# B&R Automation Studio project ControlPLC_DataDistribution (part 5)

#### Main.st - Init, cyclic, exit code
```iecst
PROGRAM _INIT

	Name := 'Print Job Management';

	// Restore current print job management information from permanent memory.
	gPrintJobManagement.currentState := Nonvolatile;

	subscribePLCOpen( gPrintJobManagement.commands.updateLayerNumber, Name, task.command.updateCurrentLayer, task.internal.PLCOpen);

	subscribePLCOpen( gPrintJobManagement.commands.validatePrintFile, Name, task.command.validatePrintFile, task.internal.PLCOpen);

	subscribePLCOpen( gSystemRecipeApi.events.buildInfoLoaded, Name, task.command.validatePrintFile, task.internal.PLCOpen);
	subscribePLCOpen( gPrintJobManagement.commands.resetPrintInfo, Name, task.command.resetPrintInfo, task.internal.PLCOpen);

	registerStateBool( gPrintJobManagement.status.buildInfoValid, 'Build Info Loaded', task.status.buildInfoValid);

	//REASONS FOR INVALID BUILD FILE
	registerStateBool( gPrintJobManagement.status.buildInfoInvalid, 'Build Name Invalid', task.status.buildInfoInvalidReasons.invalidBuildName);
	registerStateBool( gPrintJobManagement.status.buildInfoInvalid, 'Num Layers Invalid', task.status.buildInfoInvalidReasons.invalidNumLayers);
	registerStateBool( gPrintJobManagement.status.buildInfoInvalid, 'Layer Height Invalid', task.status.buildInfoInvalidReasons.invalidLayerHeight);
	registerStateBool( gPrintJobManagement.status.buildInfoInvalid, 'Platform ID Invalid', task.status.buildInfoInvalidReasons.invalidPlatformID);
	registerStateBool( gPrintJobManagement.status.buildInfoInvalid, 'Machine Name Invalid', task.status.buildInfoInvalidReasons.invalidMachineName);
	registerStateBool( gPrintJobManagement.status.buildInfoInvalid, 'Pixel Map Ver. Invalid', task.status.buildInfoInvalidReasons.invalidPixelMapVersion);
	//registerStateBool( gPrintJobManagement.status.buildInfoInvalid, 'Pixel Usage Invalid', task.status.buildInfoInvalidReasons.invalidPixelUsage);

	//	registerStateBool( gPrintJobManagement.status.buildInfoInvalid, 'Workspace Boundaries Invalid', task.status.buildInfoInvalidReasons.invalidWorkspace);	 //TODO ADD BACK WHEN BUILD INFO FILE HAS THIS

	registerStateBool( gPrintJobManagement.status.buildInfoInvalid, 'PCI File Invalid', task.status.buildInfoInvalidReasons.invalidPrintConfigInstruction);

	gConfiguration.machineIdentity.machineName := 'DP12';
	gConfiguration.machineIdentity.machineNumber := 12;

	//SIM helper for bootup to set some non vol
	IF gSimulation THEN
		//gConfiguration.machineIdentity.factoryName := 'VulcanOne';
		//gConfiguration.machineIdentity.factoryNumber := FACTORY_VULCAN_ONE;
		//gConfiguration.machineIdentity.machineGeneration := MACHINE_GENERATION_GEN3;
			gConfiguration.machineIdentity.machineName := 'DP12';
		//gConfiguration.machineIdentity.machineType := MACHINE_TYPE_PRINTER;
		//	gConfiguration.machineIdentity.machineNumber := 13;

	END_IF

END_PROGRAM

PROGRAM _CYCLIC

	//Copy current state to non-volatile memory.
	Nonvolatile := gPrintJobManagement.currentState;
	dCurrentState ACCESS ADR(gPrintJobManagement.currentState);

	task.status.ready := TRUE;

	IF gSimulation THEN
		SimulateIO;
	END_IF
	/////////////////////////////////////////////////////////////////////////////////////////////////
	//COMMANDS
	//validate build info file
	//check if ready for printing
	//increment layer number

	//Cyclically this task also manages the part height and parameters related to the build info file
	/////////////////////////////////////////////////////////////////////////////////////////////////

	IF task.status.ready THEN

		IF task.internal.localLockout THEN

		ELSIF task.command.validatePrintFile THEN

			task.internal.newCommand := TRUE;
			task.status.statusMessage := 'Validating Build Info File';
			task.status.state := STATE_VALIDATING_BUILD_INFO;

		ELSIF task.command.updateCurrentLayer THEN

			task.internal.newCommand := TRUE;
			task.status.statusMessage := 'Updating Layer Number';
			task.status.state := STATE_UPDATE_LAYER_NUMBER;

		END_IF

	ELSE

		IF NOT allZero( ADR(task.command), SIZEOF(task.command)) THEN
			//vfAlarmEdgeSnippet(gPrintJobManagement.alarms.components, gPrintJobManagement.alarms.COMMAND_BEFORE_READY, 'Print Job Manager');
		END_IF

		task.internal.PLCOpen.status := PRINT_JOB_MANAGER_ERROR;
		task.status.state := STATE_NOT_READY;
		task.internal.localLockout := FALSE;

	END_IF

	///////////////////////////////////////////////////////////////
	// Handle any canceled commands that are required
	///////////////////////////////////////////////////////////////
	IF task.internal.newCommand THEN

		// TODO: Log state changes
		//		task.internal.abortedStep := task.status.sequence;
		//		task.internal.abortedState := task.internal.previousState;

		task.status.sequence := SEQUENCE_IDLE;

		// If a new command came into the system, abort any PLCOpen commands that were active.
		// If the command came from PLCOpen FirstPass will be true and it will not abort it
		atnPLCOpenAbort(task.internal.PLCOpen);

	END_IF

	CASE task.status.state OF

		STATE_NOT_READY:

			task.status.sequence := SEQUENCE_IDLE;

			task.status.statusMessage := 'Print job manager is not in ready state';

			IF task.status.ready THEN

				task.status.state := STATE_READY;

				task.status.statusMessage := 'Print job manager is in ready state';

			END_IF

		STATE_READY:

			task.status.sequence := SEQUENCE_IDLE;
			task.internal.localLockout := FALSE;

		STATE_RESETTING_PRINT_INFO:

			CASE task.status.sequence OF

				SEQUENCE_ERROR:
					task.status.statusMessage := 'Error resetting print data';

					//Handle Error
					task.internal.PLCOpen.status := PRINT_JOB_MANAGER_ERROR;
					task.status.state := STATE_READY;

				SEQUENCE_DONE:
					task.status.statusMessage := 'Print Data has been Reset';

					//Handle Done
					task.internal.PLCOpen.status := ERR_OK;
					task.status.state := STATE_READY;

				SEQUENCE_IDLE:

					task.status.statusMessage := 'Resetting Print Data';
					task.status.sequence := SEQUENCE_ABORT_DISTRIBUTION;

				ELSE

					ResetPrintInfoSubsequence;

			END_CASE

		STATE_UPDATE_LAYER_NUMBER:

			dCurrentState.currentLayerNumber := gPrintJobManagement.currentState.nextLayerNumber;

			Nonvolatile.currentLayerNumber := dCurrentState.currentLayerNumber;

			// Convert the current layer number to a string with the "nnnnn" format, adding required leading 0s.
			brsitoa(dCurrentState.currentLayerNumber, ADR(layerNumberValue_string));
			IF (dCurrentState.currentLayerNumber > 9999) THEN
				layerNumber_string := '';
			ELSIF (dCurrentState.currentLayerNumber > 999) THEN
				layerNumber_string := '0';
			ELSIF (dCurrentState.currentLayerNumber > 99) THEN
				layerNumber_string := '00';
			ELSIF (dCurrentState.currentLayerNumber > 9) THEN
				layerNumber_string := '000';
			ELSE
				layerNumber_string := '0000';
			END_IF
			brsstrcat(ADR(layerNumber_string), ADR(layerNumberValue_string));

			// Format the complete layer filename for the G-code (CNC) motion control file.
			layerFilename_GCode := Nonvolatile.baseFilename;
			brsstrcat(ADR(layerFilename_GCode), ADR('_L'));
			brsstrcat(ADR(layerFilename_GCode), ADR(layerNumber_string));
			brsstrcat(ADR(layerFilename_GCode), ADR('_GCode.cnc'));
			task.status.currentLayerGCodeFilename := layerFilename_GCode;

			task.internal.PLCOpen.status := ERR_OK;
			task.status.state := STATE_READY;

		STATE_VALIDATING_BUILD_INFO:

			CASE task.status.sequence OF

				SEQUENCE_ERROR:
					task.status.statusMessage := 'Error Validating Print Files';

					//Handle Error
					task.internal.PLCOpen.status := PRINT_JOB_MANAGER_ERROR;
					task.status.state := STATE_READY;

				SEQUENCE_DONE:
					task.status.statusMessage := 'Validating Print files finished';
					gPrintJobManagement.status.buildInfoValidCheck := TRUE;
					//Handle Done
					task.internal.PLCOpen.status := ERR_OK;
					task.status.state := STATE_READY;

				SEQUENCE_IDLE:

					task.status.statusMessage := 'Print File validation started';
					task.status.sequence := SEQUENCE_READ_BUILD_INFO;

				ELSE

					ValidateBuildFileSubsequence;
			END_CASE

	END_CASE

	//get reason that might occur outside of the sequence
	task.status.buildInfoError := stateTrueStatus( gPrintJobManagement.status.buildInfoInvalid, ADR( task.status.buildInfoErrorStatus ), SIZEOF(task.status.buildInfoErrorStatus));

	//---------------------------------------------------------------------------
	// Repopulate layer gcode file name if PLC restarted.
	//---------------------------------------------------------------------------

	IF (task.status.currentLayerGCodeFilename = '')  THEN

		// Convert the current layer number to a string with the "nnnnn" format, adding required leading 0s.
		brsitoa(dCurrentState.currentLayerNumber, ADR(layerNumberValue_string));
		IF (dCurrentState.currentLayerNumber > 9999) THEN
			layerNumber_string := '';
		ELSIF (dCurrentState.currentLayerNumber > 999) THEN
			layerNumber_string := '0';
		ELSIF (dCurrentState.currentLayerNumber > 99) THEN
			layerNumber_string := '00';
		ELSIF (dCurrentState.currentLayerNumber > 9) THEN
			layerNumber_string := '000';
		ELSE
			layerNumber_string := '0000';
		END_IF
		brsstrcat(ADR(layerNumber_string), ADR(layerNumberValue_string));

		// Format the complete layer filename for the G-code (CNC) motion control file.
		layerFilename_GCode := Nonvolatile.baseFilename;
		brsstrcat(ADR(layerFilename_GCode), ADR('_L'));
		brsstrcat(ADR(layerFilename_GCode), ADR(layerNumber_string));
		brsstrcat(ADR(layerFilename_GCode), ADR('_GCode.cnc'));
		task.status.currentLayerGCodeFilename := layerFilename_GCode;

	END_IF

	//RESET COMMANDS
	brsmemset(ADR(task.command), 0, SIZEOF(task.command));
	task.internal.newCommand := FALSE;

	task.internal.newCommand := 0;

	command();
	IF command.Done OR command.Error OR command.Aborted THEN
		command.Execute := FALSE;
	END_IF

	logStateChange_0.LoggerName := 'App';
	logStateChange_0.ModuleName := Name;
	logStateChange_0.State 		:= task.status.state;
	logStateChange_0.StateName 	:= task.status.statusMessage;
	logStateChange_0();

	logSeqChange_0.LoggerName 	:= 'App';
	logSeqChange_0.ModuleName 	:= Name;
	//	logSeqChange_0.State		:= task.status.sequence;
	//	logSeqChange_0.StateName	:= task.status.statusMessage;
	//	logSeqChange_0();

	// ---------------------------------------------------------------------------
	// Call ATN FUB
	// ---------------------------------------------------------------------------

	//task.status.buildInfoValid := stateAllFalse( gPrintJobManagement.status.buildInfoInvalid, TRUE);

	gPrintJobManagement.status.currentLayerGCodeFilename := task.status.currentLayerGCodeFilename;

END_PROGRAM

PROGRAM _EXIT

END_PROGRAM
```

#### Types.typ - Local data types
```iecst
TYPE
	test_typ : 	STRUCT
		command : testCommand_typ;
	END_STRUCT;
	testCommand_typ : 	STRUCT
		induceCurrentLayerToEleven : BOOL;
		assertDOMS : BOOL;
		assertRegularPlate : BOOL;
	END_STRUCT;
	Configuration_typ : 	STRUCT
		BUILD_PLATE_THICKNESS_MAX_MM : REAL;
		BLADE_OFFSET_MAX_MM : REAL;
		FOCAL_OFFSET_MAX_MM : REAL;
		FOCAL_OFFSET_MIN_MM : REAL;
		FOCAL_OFFSET_MM : REAL;
		OPTICS_BOX_REVISION : USINT;
		BLADE_OFFSET_MM : REAL;
		ENCODER_TICK_WIDTH : REAL;
		MAX_LASER_COUNT : UINT;
		LASER_LINE_ANGLE : REAL;
		HEAD_CENTER_OFFSET : REAL;
		LASER_SPACING : REAL;
		MIN_LASER_WATTS : REAL;
		MAX_LASER_WATTS : REAL;
	END_STRUCT;
	IO_typ : 	STRUCT
		_ : USINT;
	END_STRUCT;
	localInterface_typ : 	STRUCT
		command : localInterfaceCommand_typ;
		parameters : localInterfaceParameter_typ;
		status : localInterfaceStatus_typ;
		internal : localInterfaceInternal_typ;
	END_STRUCT;
	localInterfaceCommand_typ : 	STRUCT
		updateCurrentLayer : BOOL;
		validatePrintFile : BOOL;
		checkReadyForPrinting : BOOL;
		resetLayerNumberToZero : BOOL;
		restartAtSpecifiedLayer : BOOL;
		setBuildPlateThickness : BOOL;
		setFocalOffset : BOOL;
		publishConfigurationData : BOOL;
		setRecoaterOffset : BOOL;
		resetPrintInfo : BOOL;
		bladeOffsetClr : BOOL;
		bladeOffsetPlusTen : BOOL;
		bladeOffsetMinusTen : BOOL;
		setThicknessDOMS : BOOL;
		clearThicknessDOMS : BOOL;
		resetPlateType : BOOL;
		enableLOP : BOOL;
		disableLOP : BOOL;
		calculateRemainingPrintTime : BOOL;
		coolingDelay : BOOL;
	END_STRUCT;
	localInterfaceParameter_typ : 	STRUCT
		layerToDistribute : UINT;
		printJobLayer : UINT;
		startingLayerNumber : UDINT;
	END_STRUCT;
	localInterfaceInternal_typ : 	STRUCT
		PLCOpenConfigData : AtnPlcOpenStatus;
		PLCOpen : AtnPlcOpenStatus;
		checkPixelUsage : AtnPLCOpen;
		previousState : STATE;
		newCommand : BOOL;
		localLockout : BOOL;
		subSystemStatus : ARRAY[0..10]OF STRING[80];
		remapPixels : AtnPLCOpen;
	END_STRUCT;
	localInterfaceStatus_typ : 	STRUCT
		currentLayerGCodeFilename : STRING[255];
		recoaterOffsetInvalid : BOOL;
		focalOffset : REAL;
		recoaterOffset : REAL;
		buildPlateThicknessInvalid : BOOL;
		buildPlateThickness : REAL;
		buildInfoValid : BOOL;
		buildInfoNotInvalid : BOOL;
		buildInfoError : BOOL;
		distributionTimeout : BOOL;
		buildInfoErrorStatus : ARRAY[0..19]OF STRING[80];
		ready : BOOL;
		sequence : SEQUENCE;
		statusMessage : STRING[vfALARMS_MAX_SNIPPET_STR_LENGTH];
		state : STATE;
		buildInfoInvalidReasons : buildInfoInvalidReasons_typ;
	END_STRUCT;
	SEQUENCE :
		(
		SEQUENCE_IDLE,
		SEQUENCE_DONE,
		SEQUENCE_ERROR,
		SEQUENCE_READ_BUILD_INFO,
		SEQUENCE_CHECK_PIXEL_USAGE,
		SEQUENCE_DO_PIXEL_MAP,
		SEQUENCE_CHECK_LASERS,
		SEQUENCE_CHECK_PUMPS,
		SEQUENCE_CHECK_O2_LEVELS,
		SEQUENCE_CHECK_PNEUMATIC_SUPPLY,
		SEQUENCE_CHECK_AXES_STATE,
		SEQUENCE_CHECK_RECOATER_POS,
		SEQUENCE_CHECK_LIFT_POS,
		SEQUENCE_CHECK_LAYER_NUMBER,
		SEQUENCE_CHECK_CAMERA,
		SEQUENCE_ASK_IF_OK_TO_RESET,
		SEQUENCE_CLEAR_DATA,
		SEQUENCE_ABORT_DISTRIBUTION
		);
	STATE :
		(
		STATE_READY,
		STATE_NOT_READY,
		STATE_CHECKING_PRINT_READY,
		STATE_UPDATE_LAYER_NUMBER,
		STATE_VALIDATING_BUILD_INFO,
		STATE_SET_BUILD_PLATE_THICKNESS,
		STATE_COOLING_DELAY,
		STATE_SET_FOCAL_OFFSET,
		STATE_SET_DOMS_THICKNESS,
		STATE_SET_RECOATER_OFFSET,
		STATE_RESETTING_PRINT_INFO,
		STATE_ERROR
		);
	buildInfoInvalidReasons_typ : 	STRUCT
		invalidPixelUsage : BOOL;
		invalidPixelMapVersion : BOOL;
		invalidMachineName : BOOL;
		invalidPlatformID : BOOL;
		invalidLayerHeight : BOOL;
		invalidNumLayers : BOOL;
		invalidBuildName : BOOL;
		invalidToolpath : BOOL;
		invalidWorkspace : BOOL;
		invalidPlateOrigin : BOOL;
		invalidPrintConfigInstruction : BOOL;
	END_STRUCT;
END_TYPE
```

#### SubSequence.st
```iecst
ACTION ValidateBuildFileSubsequence:

	CASE task.status.sequence OF

		SEQUENCE_READ_BUILD_INFO:

			task.status.statusMessage := 'Checking build info contents';

			// NOTES:====================================================
			// base_filename must be 13 charaters long (e.g. VF-00001-0001)
			// build_layout and print_number must be > 0
			// num_layers must be > 0
			// layer_height must be within established range
			// PLATFORM_MEDIUM_400x600 is not currently supported
			// PrinterInfo.name must match the machineIdentity.machineName setting

			task.status.buildInfoInvalidReasons.invalidBuildName := (gBuildInformation.build_layout = 0) OR (gBuildInformation.print_number = 0) OR (brsstrlen(ADR(gBuildInformation.base_filename)) <> 13);
			task.status.buildInfoInvalidReasons.invalidNumLayers := (gBuildInformation.num_layers = 0);
			task.status.buildInfoInvalidReasons.invalidLayerHeight := (gBuildInformation.layer_height < MIN_LAYER_HEIGHT) OR (gBuildInformation.layer_height > MAX_LAYER_HEIGHT);
			task.status.buildInfoInvalidReasons.invalidPlatformID := (gBuildInformation.platform_id <> PLATFORM_SMALL_200x600) AND (gBuildInformation.platform_id <> PLATFORM_LARGE_600x600);
			task.status.buildInfoInvalidReasons.invalidMachineName := (brsstrcmp(ADR(gBuildInformation.BuildInstanceInfo.PrinterInfo.name), ADR(gConfiguration.machineIdentity.machineName)) <> 0);

			//task.status.buildInfoInvalidReasons.invalidPrintConfigInstruction := NOT(gPrintProcessConfig.MachineName = gConfiguration.machineIdentity.machineName) OR NOT(gPrintProcessConfig.FileFormatVersion = gPrintJobManagement.currentState.PCIFileFormatVersion);

			//because if nothing exists in nonvolatile then this will never work
			IF Nonvolatile.pixelMapFileVersion = 0 THEN
				Nonvolatile.pixelMapFileVersion := 1;
			END_IF

				task.status.buildInfoValid := TRUE;
				gPrintJobManagement.currentState.buildInfoCheckValid := task.status.buildInfoValid;
				// If the BuildInfo file is different from the one that was previously running, reset to layer zero to start a new print.
				(*	IF (gBuildInformation.build_layout <> dCurrentState.buildLayout)
				OR (gBuildInformation.print_number <> dCurrentState.printNumber)
				OR (gBuildInformation.layer_height <> dCurrentState.layerHeight) THEN

				task.command.resetLayerNumberToZero := TRUE;//todo
				ELSE *)

				//populate print info
				dCurrentState.baseFilename := gBuildInformation.base_filename;
				dCurrentState.buildIteration := gBuildInformation.build_iter;
				dCurrentState.buildLayout := gBuildInformation.build_layout;
				dCurrentState.printNumber := gBuildInformation.print_number;
				dCurrentState.numberOfLayers := gBuildInformation.num_layers;
				dCurrentState.layerHeight := gBuildInformation.layer_height;
				//dCurrentState.buildPlatform := PLATFORM_LARGE_600x600;//fixed value ignore BD
				dCurrentState.description := gBuildInformation.description;
				dCurrentState.author := gBuildInformation.author;
				dCurrentState.printOwner := gBuildInformation.print_owner;

				task.status.sequence := SEQUENCE_DONE;

	END_CASE

END_ACTION

ACTION ResetPrintInfoSubsequence:

	CASE task.status.sequence OF

		SEQUENCE_ABORT_DISTRIBUTION:

			executeCommand(gBuildDistributorApi.commands.abortDistribution);
			task.status.sequence := SEQUENCE_CLEAR_DATA;

		SEQUENCE_CLEAR_DATA:

			task.status.sequence := SEQUENCE_DONE;
	END_CASE

	END_ACTION
```

#### Simulation.st
```iecst
ACTION SimulateIO:

	//used in the electrode test case -> electrode only enable if layer 10 or more
	IF test.command.induceCurrentLayerToEleven THEN
		test.command.induceCurrentLayerToEleven := FALSE;
		gPrintJobManagement.currentState.currentLayerNumber := 11;
		gPrintJobManagement.currentState.lastPrintedLayerNumber := 10;
		gPrintJobManagement.currentState.lastRecoatedLayerNumber := 10;
	END_IF

END_ACTION
```

### Program Logical/DataManagement/PrintJobManagement/BuildDistributor (IEC)

#### Main.st - Init, cyclic, exit code
```iecst
PROGRAM _INIT

	Name := 'Build Distributor';

	//direct commands to operate the chiller
	subscribePLCOpenWithParameters ( gBuildDistributorApi.commands.startDistribution, Name, ADR(task.parameters.layerNumberToDistribute), SIZEOF(task.parameters.layerNumberToDistribute), task.command.startDistribution, task.internal.PLCOpen);
	subscribePLCOpen( gBuildDistributorApi.commands.distributeLayerFile, Name, task.command.distributeLayerFile, task.internal.PLCOpen );
	subscribePLCOpenWithParameters ( gBuildDistributorApi.commands.abortDistribution, Name, 0, 0, task.command.abortDistribution, task.internal.PLCOpen);

	//other systems can monitor this state
	registerStateBool( gBuildDistributorApi.status.subsystemsReady, Name, task.status.buildDistributorConnected);

END_PROGRAM

PROGRAM _CYCLIC

	//Call piper interface
	PiperModuleInterface;

	///////////////////////////////////////////////////////////////
	//API:
	//	Requires:
	//	-
	//	Commands:
	//	-takePrescan
	//	-takePostscan
	//  -takeManual
	//	Inhbits:
	//	-

	//  State Monitoring
	//  -
	///////////////////////////////////////////////////////////////

	//Heartbeat set and monitor
	task.internal.heartbeatTimer.PT := T#1s;
	task.internal.heartbeatTimer.IN := NOT(task.internal.heartbeatTimer.Q);
	IF (task.internal.heartbeatTimer.Q) THEN
		gOpcData_ToBuildPC.Heartbeat := gOpcData_ToBuildPC.Heartbeat + 1;
		IF (gOpcData_FromBuildPC.Heartbeat <> task.internal.lastHeartbeatReceived) THEN
			task.internal.lastHeartbeatReceived := gOpcData_FromBuildPC.Heartbeat;
			task.status.buildDistributorConnected := TRUE;
			task.status.missedHeartbeats := 0;
		ELSE
			task.status.missedHeartbeats := task.status.missedHeartbeats + 1;
		END_IF
	END_IF
	task.internal.heartbeatTimer();

	//timeout after 3 missed heartbeats
	IF task.status.missedHeartbeats > 10 THEN
		task.status.buildDistributorConnected := FALSE;
	END_IF

	//Reset signals if data distributor disconnects
	IF NOT(task.status.buildDistributorConnected) THEN
		gOpcData_ToBuildPC.RequestAbortDistribution := FALSE;
		gOpcData_ToBuildPC.RequestPauseDistribution := FALSE;
		gOpcData_ToBuildPC.RequestStartDistribution := FALSE;
		gOpcData_ToBuildPC.PrintingActive := FALSE;
		gOpcData_ToBuildPC.RequestBuildInfo := FALSE;
	END_IF

	//ADD LATER TODO
	//	vfAlarmPersistent(gVisionApi.alarms.components, gVisionApi.alarms.VISION_HEARTBEAT_LOST_AL1200, NOT(task.status.visionAppConnected));

	//ready to handle commands
	task.status.ready := stateTrueStatus( gBuildDistributorApi.status.subsystemsReady, ADR(task.internal.subSystemStatus), SIZEOF(task.internal.subSystemStatus) );

	IF NOT task.status.ready THEN
		stateStatus( gBuildDistributorApi.status.subsystemsReady, ADR(task.internal.subSystemStatus), SIZEOF(task.internal.subSystemStatus) );
	ELSE
		task.internal.subSystemStatus[0] := 'Ready';
	END_IF

	///////////////////////////////////////////////////////////////
	//Handle interpreting commands that do not require STATE_READY
	///////////////////////////////////////////////////////////////
	IF task.status.ready THEN

		//NOTE: Commands that just turn ON/OFF IO CAN happen in the command translation
		IF task.command.startDistribution THEN
			task.internal.newCommand := 1;

			task.status.sequence := SEQUENCE_IDLE;
			task.status.state := STATE_START_DISTRIBUTION;
			task.status.statusMessage := 'Starting Distribution';

		ELSIF task.command.distributeLayerFile THEN
			task.internal.newCommand := 1;
			task.status.sequence := SEQUENCE_IDLE;
			task.status.state := STATE_DISTRIBUTE_LAYER_FILE;
			task.status.statusMessage := 'Distributing Layer File';

		ELSIF task.command.abortDistribution THEN
			task.internal.newCommand := 1;
			task.status.sequence := SEQUENCE_IDLE;
			task.status.state := STATE_ABORT_DISTRIBUTION;
			task.status.statusMessage := 'Aborting Distribution';

		END_IF

	ELSE
		task.internal.PLCOpen.status := BUILD_DISTRIBUTOR_ERROR;
		task.status.state := STATE_NOT_READY;
		task.internal.localLockout := FALSE;
	END_IF

	///////////////////////////////////////////////////////////////
	//Handle any canceled commands that are required
	///////////////////////////////////////////////////////////////
	IF task.internal.newCommand THEN

		//TODO: Log state changes
		//		task.internal.abortedStep := task.status.sequence;
		//		task.internal.abortedState := task.internal.previousState;

		//If a new command came into the system, abort any PLCOpen commands that were active.
		// If the command came from PLCOpen FirstPass will be true and it will not abort it
		atnPLCOpenAbort(task.internal.PLCOpen);

	END_IF

	///////////////////////////////////////////////////////////////
	//Handle any Commands that do not require state.
	///////////////////////////////////////////////////////////////

	///////////////////////////////////////////////////////////////
	//Handle the current state
	///////////////////////////////////////////////////////////////
	CASE task.status.state OF

		STATE_NOT_READY:

			task.status.sequence := SEQUENCE_IDLE;
			task.status.statusMessage := 'Build Distributor is NOT ready';
			gOpcData_ToBuildPC.RequestBuildInfo := FALSE;

			IF task.status.ready THEN
				task.status.state := STATE_READY;
				task.status.statusMessage := 'Build Distributor is ready';
			END_IF

		STATE_READY:

			task.status.sequence := SEQUENCE_IDLE;
			task.internal.localLockout := FALSE;
			gOpcData_ToBuildPC.RequestBuildInfo := FALSE;

		STATE_START_DISTRIBUTION:

			CASE task.status.sequence OF

				SEQUENCE_ERROR:
					task.status.statusMessage := 'Start Distribution ERROR';
					task.internal.PLCOpen.status := BUILD_DISTRIBUTOR_ERROR;
					task.status.state := STATE_READY;

				SEQUENCE_DONE:
					task.status.statusMessage := 'Start Distribution COMPLETE';
					task.internal.PLCOpen.status := ERR_OK;
					task.status.state := STATE_READY;

				SEQUENCE_IDLE:
					task.status.statusMessage := 'Start Distribution busy...';
					task.status.sequence := SEQUENCE_EXECUTE_START_DIST;

				ELSE

					StartDistributionSubSequence;

			END_CASE

		STATE_DISTRIBUTE_LAYER_FILE:

			CASE task.status.sequence OF

				SEQUENCE_ERROR:
					task.status.statusMessage := 'Distribute Layer ERROR';
					task.internal.PLCOpen.status := BUILD_DISTRIBUTOR_ERROR;
					task.status.state := STATE_READY;

				SEQUENCE_DONE:
					task.status.statusMessage := 'Distribute Layer COMPLETE';
					task.internal.PLCOpen.status := ERR_OK;
					task.status.state := STATE_READY;

				SEQUENCE_IDLE:
					task.status.statusMessage := 'Distribute Layer busy...';
					task.status.sequence := SEQUENCE_EXECUTE_GET_LAYER_FILES;

				ELSE

					DistributeLayerFileSubSequence;

			END_CASE

		STATE_ABORT_DISTRIBUTION:

			task.status.statusMessage := 'aborting distribution';

			IF task.status.buildDistributorConnected THEN
				//gPrint Job management files
				gOpcData_ToBuildPC.RequestAbortDistribution := TRUE;
				gOpcData_ToBuildPC.RequestPauseDistribution := FALSE;
				gOpcData_ToBuildPC.RequestStartDistribution := FALSE;
				gOpcData_ToBuildPC.PrintingActive := FALSE;
				gOpcData_ToBuildPC.RequestBuildInfo := FALSE;

				IF (gOpcData_FromBuildPC.DistributionAborted) THEN
					gOpcData_ToBuildPC.RequestAbortDistribution := FALSE;

					//brsmemset( ADR(gPrintProcessConfig), 0, SIZEOF(gPrintProcessConfig) ); Not deleting. Keep last know value on Abort
					gPrintProcessConfigLoaded := FALSE;

					task.status.statusMessage := 'aborting complete';
					task.internal.PLCOpen.status := ERR_OK;
					task.status.state := STATE_READY;

				END_IF

			ELSE
				task.status.statusMessage := 'BD not connected';
				gOpcData_ToBuildPC.RequestAbortDistribution := FALSE;
				task.status.state := STATE_READY;
				task.internal.PLCOpen.status := ERR_OK;

			END_IF

	END_CASE

	///////////////////////////////////////////////////////////////
	//Update Statuses
	///////////////////////////////////////////////////////////////

	///////////////////////////////////////////////////////////////
	//Call all PLCOpen function blocks
	///////////////////////////////////////////////////////////////
	task.internal.fbTON_DistributionDelay();
	task.internal.fbTON_DistributionDelay.IN := FALSE;

	task.internal.atnPLCOpenCommand();
	task.internal.atnPLCOpenCommand.Execute := FALSE;

	task.internal.atnPLCOpenCommandParameters();
	task.internal.atnPLCOpenCommandParameters.Execute := FALSE;

	task.internal.distributorTimeout();
	task.internal.distributorTimeout.IN := FALSE;

	task.internal.distributionRecoveryTimer();
	task.internal.distributionRecoveryTimer.IN := FALSE;

	///////////////////////////////////////////////////////////////
	//Reset all commands to ensure they don't get buffered
	///////////////////////////////////////////////////////////////
	task.command.distributeLayerFile := 0;
	task.command.startDistribution := 0;
	task.command.abortDistribution := 0;
	task.internal.newCommand := 0;

	task.internal.waitToRetry();
	task.internal.waitToRetry.IN := FALSE;

	logStateChange_0.LoggerName := 'App';
	logStateChange_0.ModuleName := Name;
	logStateChange_0.State 		:= task.status.state;
	logStateChange_0.StateName 	:= task.status.statusMessage;
	logStateChange_0();

	logSeqChange_0.LoggerName 	:= 'App';
	logSeqChange_0.ModuleName 	:= Name;
	logSeqChange_0.State		:= task.status.sequence;
	logSeqChange_0.StateName	:= task.status.statusMessage;
	logSeqChange_0();

	//Keep track of the previous state
	task.internal.previousState := task.status.state;

	///////////////////////////////////////////////////////////////
	//Simulation
	///////////////////////////////////////////////////////////////
	IF gSimulation THEN
		SimulateIO;
	END_IF

END_PROGRAM

PROGRAM _EXIT
		(* Insert code here *)

END_PROGRAM
```

#### PiperInterface.st
```iecst
ACTION PiperModuleInterface:

	//Give this module a name so it is easier to debug
	ModuleInterface.ModuleName:=	Name;

	//Add a module to the Piper
	Module.ModuleInterface:=	ADR(ModuleInterface);
	Module.Piper:= 	ADR(gMachine);
	Module();

	// Handle any machine states that this module needs to respond to
	CASE ModuleInterface.PiperState OF
//		MACH_ST_BOOTING:
//		MACH_ST_CLEARING:
//		MACH_ST_STOPPED:
		MACH_ST_STARTING:

			ModuleInterface.ModuleResponse:=	ModuleInterface.PiperState;

			(*//sample piper integration

			//for when sequence is required for substate transition
			CASE ModuleInterface.PiperSubState OF

				0:

					//only need the chiller for printing but not other operations
					CASE gMachineState.operation OF

						MACHINE_OPERATIONS_PRINT_LAYER:
							ModuleInterface.ModuleSubStateRequest := SUB_STATE_CHECK_CHILLER;

						ELSE
							ModuleInterface.ModuleResponse:=	ModuleInterface.PiperState;

					END_CASE

				SUB_STATE_CHECK_CHILLER:

					//should be an edge command
					task.command.startChiller := TRUE;

					ModuleInterface.ModuleStatus := 'waiting chiller';

					IF task.status.chillerIsRunning THEN
						ModuleInterface.ModuleResponse:=	ModuleInterface.PiperState;
					END_IF

			END_CASE

			*)

//		MACH_ST_IDLE:
//		MACH_ST_SUSPENDED:
//		MACH_ST_EXECUTE:
//		MACH_ST_STOPPING:
//		MACH_ST_ABORTING:
//		MACH_ST_ABORTED:
//		MACH_ST_HOLDING:
//		MACH_ST_HELD:
//		MACH_ST_UNHOLDING:
//		MACH_ST_SUSPENDING:
//		MACH_ST_UNSUSPENDING:
//		MACH_ST_RESETTING:
//		MACH_ST_COMPLETING:
//		MACH_ST_COMPLETE:

		MACH_ST_BYPASSED:

		ELSE
			ModuleInterface.ModuleResponse:=	ModuleInterface.PiperState;

	END_CASE

	//for turning commands to edges to work with piper
	(*
	//Turn level commands to edges
	EdgePosArray( ADR(piperCommands), ADR(_piperCommands), ADR(task.command), SIZEOF(task.command) );
	brsmemset( ADR(piperCommands), 0, SIZEOF(piperCommands) );
	*)

END_ACTION
```

#### SubSequence.st
```iecst
// Start connection to build distributor and distribute the starting files
ACTION StartDistributionSubSequence:

	CASE task.status.sequence OF

		SEQUENCE_EXECUTE_START_DIST:

			task.status.sequence := SEQUENCE_REQUEST_BUILD_INFO;

		SEQUENCE_REQUEST_BUILD_INFO:

			task.status.statusMessage := 'ask for build info file';

			//gPrint Job management files
			gOpcData_ToBuildPC.RequestAbortDistribution := FALSE;
			gOpcData_ToBuildPC.RequestPauseDistribution := FALSE;
			gOpcData_ToBuildPC.RequestStartDistribution := FALSE;
			gOpcData_ToBuildPC.PrintingActive := FALSE;
			gOpcData_ToBuildPC.RequestBuildInfo := TRUE;

			//load the last file you had saved, if its 0 get layer 1
			gOpcData_ToBuildPC.CurrentPrintLayer := gPrintJobManagement.currentState.currentLayerNumber;
			IF (gOpcData_ToBuildPC.CurrentPrintLayer = 0) THEN
				gOpcData_ToBuildPC.CurrentPrintLayer := 1;
			END_IF

			task.status.sequence := SEQUENCE_BUILD_INFO_READY;

		SEQUENCE_BUILD_INFO_READY:

			IF (gOpcData_FromBuildPC.BuildInfoReady) THEN
				gOpcData_ToBuildPC.RequestBuildInfo := FALSE;
				task.status.sequence := SEQUENCE_LOAD_PCI_FILE;
			END_IF

		SEQUENCE_LOAD_PCI_FILE:

			task.status.statusMessage := 'Loading PCI File and Verifying';

			task.internal.atnPLCOpenCommand.Command := gSystemRecipeApi.commands.loadPrintProcessConfigFile;
			task.internal.atnPLCOpenCommand.Execute := TRUE;

			IF task.internal.atnPLCOpenCommand.Done OR gPrintJobManagement.status.loadPCIFileComplete THEN
				task.status.sequence := SEQUENCE_LOAD_BUILD_FILE;
				task.internal.atnPLCOpenCommand.Execute := FALSE;
				gPrintJobManagement.status.loadPCIFileComplete := FALSE;

			ELSIF task.internal.atnPLCOpenCommand.Error THEN
				task.status.sequence := SEQUENCE_ERROR;
			END_IF

		SEQUENCE_LOAD_BUILD_FILE:
			task.status.statusMessage := 'load build info file';
			task.internal.atnPLCOpenCommand.Command := gSystemRecipeApi.commands.loadBuildInfo;
			task.internal.atnPLCOpenCommand.Execute := TRUE;

			IF task.internal.atnPLCOpenCommand.Done OR gSystemRecipeApi.status.buildInfoLoaded THEN
				task.status.sequence := SEQUENCE_CHK_BUILD_INFO_VALID;
				gSystemRecipeApi.status.buildInfoLoaded := FALSE;
				task.internal.atnPLCOpenCommand.Execute := FALSE;

			ELSIF task.internal.atnPLCOpenCommand.Error THEN
				task.status.sequence := SEQUENCE_ERROR;
			END_IF

		SEQUENCE_CHK_BUILD_INFO_VALID:
			task.status.statusMessage := 'validating build info contents';
			task.internal.atnPLCOpenCommand.Command := gPrintJobManagement.commands.validatePrintFile;
			task.internal.atnPLCOpenCommand.Execute := TRUE;

			IF task.internal.atnPLCOpenCommand.Done OR gPrintJobManagement.status.buildInfoValidCheck THEN
				task.status.sequence := SEQUENCE_DELETE_LASER_FILES;
				gPrintJobManagement.status.buildInfoValidCheck:= FALSE;
				task.internal.atnPLCOpenCommand.Execute := FALSE;
				gPrintProcessConfigLoaded := TRUE; // Set flag after validating PCI with BuildInfo File
			ELSIF task.internal.atnPLCOpenCommand.Error THEN
				task.status.sequence := SEQUENCE_ERROR;
			END_IF

		SEQUENCE_DELETE_LASER_FILES:
			task.status.statusMessage := 'delete laser files';
			task.internal.atnPLCOpenCommand.Command := gVFLCR.command.deleteLaserControlFiles;
			task.internal.atnPLCOpenCommand.Execute := TRUE;

			IF task.internal.atnPLCOpenCommand.Done THEN
				task.status.sequence := SEQUENCE_START_DISTRIBUTION;
				task.internal.atnPLCOpenCommand.Execute := FALSE;
			ELSIF task.internal.atnPLCOpenCommand.Error THEN
				task.status.sequence := SEQUENCE_ERROR;
			END_IF

		SEQUENCE_START_DISTRIBUTION:
			task.status.statusMessage := 'distribute laser files';

			gOpcData_ToBuildPC.RequestStartDistribution := TRUE;
			task.status.sequence := SEQUENCE_VERIFY_DISTRIBUTION;

		SEQUENCE_VERIFY_DISTRIBUTION:

			task.status.statusMessage := 'verifying distribution';

			IF (gOpcData_FromBuildPC.CurrentDistributionLayer = gOpcData_ToBuildPC.CurrentPrintLayer) THEN

				task.internal.lastDistributedLayerNumber := UDINT_TO_UINT(gOpcData_ToBuildPC.CurrentPrintLayer);
				gPrintJobManagement.currentState.lastDistributedLayer := task.internal.lastDistributedLayerNumber;

				task.status.sequence := SEQUENCE_SET_CURRENT_LAYER;

			END_IF

			task.internal.distributorTimeout.PT := T#30s;
			task.internal.distributorTimeout.IN := TRUE;

			IF task.internal.distributorTimeout.Q THEN
				task.status.sequence := SEQUENCE_ERROR;
			END_IF

		SEQUENCE_SET_CURRENT_LAYER:

			//this is redundant, but that command also will re-set the CNC file name
			task.status.statusMessage := 'update current layer';

			//NOT NEEDED!
			Nonvolatile.currentLayerNumber := gPrintJobManagement.currentState.currentLayerNumber;

			task.status.sequence := SEQUENCE_DISTRIBUTION_STARTED;

		SEQUENCE_DISTRIBUTION_STARTED:
			gPrintJobManagement.currentState.newBuildInfoFileLoaded := TRUE;//TODO this should be set outside?
			task.status.sequence := SEQUENCE_DONE;
	END_CASE

END_ACTION

// Distribute Layer Files to VFLCR and adjust number
ACTION DistributeLayerFileSubSequence:

	CASE task.status.sequence OF

		SEQUENCE_EXECUTE_GET_LAYER_FILES:
			task.status.sequence := SEQUENCE_SET_DESIRED_LAYER;

		SEQUENCE_CHK_BUILD_INFO:
			task.status.statusMessage := 'validating build info';
			task.internal.atnPLCOpenCommand.Command := gPrintJobManagement.commands.validatePrintFile;
			task.internal.atnPLCOpenCommand.Execute := TRUE;

			IF task.internal.atnPLCOpenCommand.Done OR gPrintJobManagement.status.buildInfoValidCheck THEN
				task.status.sequence := SEQUENCE_SET_DESIRED_LAYER;
				task.internal.atnPLCOpenCommand.Execute := FALSE;
				gPrintJobManagement.status.buildInfoValidCheck := FALSE;
			ELSIF task.internal.atnPLCOpenCommand.Error THEN

				task.status.lastErrorMessage := 'SEQUENCE_CHK_BUILD_INFO';
				task.status.sequence := SEQUENCE_ERROR;
			END_IF

		SEQUENCE_SET_DESIRED_LAYER:

			task.internal.distRetryAttempted := 0;

			task.status.statusMessage := 'set layer for distribution';
			gOpcData_ToBuildPC.CurrentPrintLayer := gPrintJobManagement.currentState.nextLayerNumber;

			//delay for parameter to go through
			task.internal.fbTON_DistributionDelay.PT := T#0.25s;
			task.internal.fbTON_DistributionDelay.IN := TRUE;
			IF task.internal.fbTON_DistributionDelay.Q THEN
				task.status.sequence := SEQUENCE_REQUEST_DISTRIBUTION;
			END_IF

		SEQUENCE_REQUEST_DISTRIBUTION:

			task.status.statusMessage := 'request distribution';
			gOpcData_ToBuildPC.PrintingActive := TRUE;
			gOpcData_ToBuildPC.RequestStartDistribution := TRUE;
			task.status.sequence := SEQUENCE_WAIT_FOR_FEEDBACK;

		SEQUENCE_WAIT_FOR_FEEDBACK:

			IF (gOpcData_FromBuildPC.CurrentDistributionLayer = gOpcData_ToBuildPC.CurrentPrintLayer) THEN
				task.status.sequence := SEQUENCE_DONE;
				gPrintJobManagement.status.distributionLayerComplete := TRUE;
			END_IF

			task.internal.distributorTimeout.IN := TRUE;
			task.internal.distributorTimeout.PT := T#20s;

			IF task.internal.distributorTimeout.Q  THEN

				IF task.internal.distRetryAttempted THEN
					task.status.sequence := SEQUENCE_ERROR;
				ELSE
					task.status.sequence := SEQUENCE_RETRY_DISTRIBUTION;
				END_IF

			END_IF

		SEQUENCE_RETRY_DISTRIBUTION:

			gOpcData_ToBuildPC.CurrentPrintLayer := 0;

			task.internal.distributionRecoveryTimer.IN := TRUE;
			task.internal.distributionRecoveryTimer.PT := T#5s;

			IF task.internal.distributionRecoveryTimer.Q THEN
				task.internal.distRetryAttempted := TRUE;
				gOpcData_ToBuildPC.CurrentPrintLayer := task.parameters.layerNumberToDistribute;
				task.status.sequence := SEQUENCE_REQUEST_DISTRIBUTION;
			END_IF

		SEQUENCE_SET_CURRENT_LAYER:

			task.status.statusMessage := 'update current layer';

			task.internal.lastDistributedLayerNumber := UDINT_TO_UINT(gOpcData_ToBuildPC.CurrentPrintLayer);
			gPrintJobManagement.currentState.lastDistributedLayer := task.internal.lastDistributedLayerNumber;

			task.internal.atnPLCOpenCommandParameters.Command := gPrintJobManagement.commands.updateLayerNumber;
			task.internal.atnPLCOpenCommandParameters.pParameters := ADR(task.internal.lastDistributedLayerNumber);
			task.internal.atnPLCOpenCommandParameters.sParameters := SIZEOF(task.internal.lastDistributedLayerNumber);
			task.internal.atnPLCOpenCommandParameters.Execute := TRUE;

			IF task.internal.atnPLCOpenCommandParameters.Done THEN
				task.status.sequence := SEQUENCE_DONE;
				task.internal.atnPLCOpenCommandParameters.Execute := FALSE;

			ELSIF task.internal.atnPLCOpenCommandParameters.Error THEN
				task.status.lastErrorMessage := 'SEQUENCE_SET_CURRENT_LAYER';

				IF NOT(task.internal.retryAttempted) THEN
					task.status.sequence := SEQUENCE_RETRY_AFTER_ERROR;
					task.status.lastErrorState := SEQUENCE_SET_CURRENT_LAYER;
				ELSE
					task.status.sequence := SEQUENCE_ERROR;
					task.internal.retryAttempted := FALSE;
				END_IF
			END_IF

		SEQUENCE_RETRY_AFTER_ERROR:

			task.internal.retryAttempted := TRUE;

			task.internal.waitToRetry.PT := T#5s;
			task.internal.waitToRetry.IN := TRUE;

			IF task.internal.waitToRetry.Q THEN
				task.status.sequence := task.status.lastErrorState;
			END_IF

	END_CASE

END_ACTION

// Abort distribution process started earlier (must be done before starting another)
ACTION AbortDistributionSubSequence:

	CASE task.status.sequence OF

		SEQUENCE_EXECUTE_ABORT_DIST:

			task.status.sequence := SEQUENCE_CHECK_DIST_READY_ABORT;

		SEQUENCE_CHECK_DIST_READY_ABORT:
			task.status.statusMessage := 'check distributor connected';
			//move this outside maybe and cyclically check for connection status and throw alarm if not connected
			IF task.status.buildDistributorConnected THEN
				task.status.sequence := SEQUENCE_REQUEST_ABORT_DIST;
			ELSE
				task.status.sequence := SEQUENCE_ERROR;
			END_IF

		SEQUENCE_REQUEST_ABORT_DIST:

			task.status.statusMessage := 'aborting distribution';

			//gPrint Job management files
			gOpcData_ToBuildPC.RequestAbortDistribution := TRUE;
			gOpcData_ToBuildPC.RequestPauseDistribution := FALSE;
			gOpcData_ToBuildPC.RequestStartDistribution := FALSE;
			gOpcData_ToBuildPC.PrintingActive := FALSE;
			gOpcData_ToBuildPC.RequestBuildInfo := FALSE;

			task.status.sequence := SEQUENCE_WAIT_DIST_ABORTED;

		SEQUENCE_WAIT_DIST_ABORTED:

			task.status.statusMessage := 'distribution aborted';

			IF (gOpcData_FromBuildPC.DistributionAborted) THEN
				gOpcData_ToBuildPC.RequestAbortDistribution := FALSE;
				task.status.sequence := SEQUENCE_DONE;;
			END_IF

	END_CASE

END_ACTION
```

### Program Logical/Infrastructure/FirstInitProg (ANSIC)

#### FirstInitProgInit.c - Initialization code
```c
/********************************************************************
 * COPYRIGHT --
 ********************************************************************
 * Program: FirstInitProg
 * File: FirstInitProgInit.c
 * Author: ScismD
 * Created: January 07, 2014
 ********************************************************************
 * Implementation of program FirstInitProg
 ********************************************************************/

// TODO: convert to ST

#include <bur/plctypes.h>

//#ifdef _DEFAULT_INCLUDES
#include <AsDefault.h>
//#endif

#include <string.h>

void _INIT FirstInitProgInit(void)
{

	gTransfer = gCyclic;

	if( strcmp(_buildDate, gRevInfo_buildDate) != 0 || gTransfer){
		gBootAfterTransfer = !gTransfer;
		gDataValid[0] = 0;
		gDataValid[1] = 0;
	}
	if(!gTransfer){
		strcpy(_buildDate, gRevInfo_buildDate);
	}

	// Check for simulation
	// This is a DevLink using a Windows share which is not supported by ARsim
	// We use this instead of Diag function to support older CPU's
	simCheckDevLink.enable = 1;
	simCheckDevLink.pDevice = (UDINT)&("SimCheck");
	simCheckDevLink.pParam = (UDINT)&("/SIP=127.0.0.1 /PROTOCOL=cifs /SHARE=testfolder /USER=max /PASSWORD=passw");

	DevLink(&simCheckDevLink);

	if (simCheckDevLink.status == ERR_NOTIMPLEMENTED) {
		gSimulation = 1;
	}

	// Initialize User Loggers
	createLogInit("Errors", 1000000, arEVENTLOG_PERSISTENCE_VOLATILE);
	createLogInit("Files", 1000000, arEVENTLOG_PERSISTENCE_VOLATILE);
	createLogInit("App", 1000000, arEVENTLOG_PERSISTENCE_VOLATILE);

	// INIT ATN Interfaces
	//-------------------------------------------------------
	atninit( &gConsole.Console, sizeof(gConsole.Console) );

	varPopulateMemberNames( "gStates", strlen(&"gStates") + 1);
	varPopulateMemberNames( "gActions", strlen(&"gActions") + 1);
	varPopulateMemberNames( "gCommands", strlen(&"gCommands") + 1);
	varPopulateMemberNames( "gVFLCR", 0 );
	varPopulateMemberNames( "gSFCControlApi", 0 );
	varPopulateMemberNames( "gAlarmApi", 0 );

	// Link file devices
	//-------------------------------------------------------

	// This is NOT done in the CPU configuration because when using CPU simulation
	// you cannot have separate file devices for simulation mode,
	// and you cannot unlink devices that were entered in the CPU configuration

	// Set up file device names
	strcpy(fileDevice[3], "PermData");
	strcpy(fileDevice[6], "PixelMapping");
	strcpy(fileDevice[7], "CurrentBuild");

	// Set up file device paths
	if (gSimulation) {
		strcpy(directory[0], "C:\\ARSimUser\\ControlPLC_Gen3");
		strcpy(directory[3], "C:\\ARSimUser\\ControlPLC_Gen3\\PermData");
		strcpy(directory[6], "C:\\ARSimUser\\ControlPLC_Gen3\\CurrentBuild");
		strcpy(directory[7], "C:\\ARSimUser\\ControlPLC_Gen3\\CurrentBuild");
	} else {
		// TODO: This won't work (nicely) with ARwin
		strcpy(directory[0], "F:\\");
		strcpy(directory[3], "F:\\PermData");
		strcpy(directory[6], "F:\\CurrentBuild");
		strcpy(directory[7], "F:\\CurrentBuild");
	}

	// Link file devices
	for (i = 0; i < NUM_FILEDEVICES; i++) {

		strcpy(parameters[i], "/DEVICE=");
		strcat(parameters[i], directory[i]);

		fileDeviceDevLink[i].enable = 1;
		fileDeviceDevLink[i].pDevice = (UDINT)&(fileDevice[i]);
		fileDeviceDevLink[i].pParam =  (UDINT)&(parameters[i]);

		DevLink(&fileDeviceDevLink[i]);

	}

	// Initialize Persisters
	//-------------------------------------------------------

	// Working variables

	// Machine configuration
	varGetVariableList((UDINT)"Configuration", (UDINT)&(gPersister[PERM_CONFIGURATION].IN.WorkingVariableList));

	// Home data
	strcpy(gPersister[PERM_HOME_DATA].IN.WorkingVariableList[0],"RestorePosition");

	// Permanent variables
	gPersister[PERM_CONFIGURATION].IN.pPersistentVariable = (UDINT)&gPermConfiguration;
	gPersister[PERM_CONFIGURATION].IN.sizeofPersistentVariable = sizeof(gPermConfiguration);

	gPersister[PERM_HOME_DATA].IN.pPersistentVariable = (UDINT)&gPermHomeData;
	gPersister[PERM_HOME_DATA].IN.sizeofPersistentVariable = sizeof(gPermHomeData);

	// DataValid and PersistFn_Init()
	for(i = 0; i < NUM_PERSISTERS; i++){
		gPersister[i].IN.pDataValid = (UDINT)&gDataValid[i];
		PersistFn_Init(&gPersister[i]);
		if(gPersister[i].OUT.STAT.Error){
			persistErrorID = gPersister[i].OUT.STAT.ErrorID;
			//vfAlarmEdgeSnippet(&gMachineAlarms.components, &gMachineAlarms.PERMMEM_PERSISTER_ERROR, gPersister[i].OUT.STAT.ErrorString);
		}
		if( gPersister[i].OUT.STAT.RequiredMemory != gPermDataSize[i]){
			gDataValid[i] = 0;
			//			vfAlarmEdgeSnippet(&gMachineAlarms.components, &gMachineAlarms.PERMMEM_PERSISTER_SIZE_CHANGED, gPersister[i].OUT.STAT.ErrorString);
		}
	}

	//-------------------------------------------------------
	// Load task configurations
	//-------------------------------------------------------

	// TODO: check retval of this varGetVariableList call and add alarm when we've exceeded max number of configs
	varGetVariableList((UDINT)"Configuration", (UDINT)&(gSplitConfig.configList));
	strcpy(gPermData[PERM_CONFIGURATION].IN.PAR.FileDevice, "PermData");
	CSVFn_Init( &gPermData[PERM_CONFIGURATION] );

	// cache split config data
	int taskIndex;
	for( taskIndex = 0; taskIndex <= CSV_MAI_VARLIST; taskIndex++ ){
		//Go through the list until there is an empty filename
		if( gSplitConfig.configList[taskIndex][0] != 0 ){

			gSplitConfig.taskCount++;

			//The taskIndex name is the filename
			strcpy(&gSplitConfig.configFilename[taskIndex], &gSplitConfig.configList[taskIndex]);

			//Put log files in a log folder
			strcpy(&gSplitConfig.logFilename[taskIndex], "logs/");
			strcat(&gSplitConfig.logFilename[taskIndex], &gSplitConfig.configList[taskIndex]);

			//Remove the data starting from the colon. ie ':Configuration'
			char *colon;
			colon = strchr(&gSplitConfig.configFilename[taskIndex], ':');
			if( colon ){
				*colon = 0;
			}
			colon = strchr(&gSplitConfig.logFilename[taskIndex], ':');
			if( colon ){
				*colon = 0;
			}

			//Append some extensions
			strcat(&gSplitConfig.configFilename[taskIndex], ".csv");
			strcat(&gSplitConfig.logFilename[taskIndex], ".csvlog");

		}
	}

	// if persister failed, reload from csv
	if (!gDataValid[PERM_CONFIGURATION]) {
		for( taskIndex = 0; taskIndex < gSplitConfig.taskCount; taskIndex++ ){

			// run all split config CSVFileMgr setup
			strcpy(&gPermData[PERM_CONFIGURATION].IN.PAR.FileName, &gSplitConfig.configFilename[taskIndex]);
			memset(&gPermData[PERM_CONFIGURATION].IN.PAR.VariableList, 0, sizeof(gPermData[PERM_CONFIGURATION].IN.PAR.VariableList));
			memcpy(&gPermData[PERM_CONFIGURATION].IN.PAR.VariableList, &gSplitConfig.configList[taskIndex], sizeof(gSplitConfig.configList[taskIndex]));
			strcpy(&gPermData[PERM_CONFIGURATION].IN.CFG.LogFileName, &gSplitConfig.logFilename[taskIndex]);

			CSVOpenFile_Init( &gPermData[PERM_CONFIGURATION] );

			if (gPermData[PERM_CONFIGURATION].OUT.STAT.Error) {

				// error, mark data invalid for this task
				gSplitConfig.taskDataValid[taskIndex] = 0;

				//Copy filename to the alarm snippet
				strcpy( alarmSnippet, gPermData[PERM_CONFIGURATION].IN.PAR.FileName );

				//This error indicates the file doesn't exist
				// We will create a template file for the user to edit.
				if( gPermData[PERM_CONFIGURATION].OUT.STAT.ErrorID == 20708 ){

					//Alert the user that the config is wrong
					//vfAlarmEdgeSnippet( &gMachineAlarms.components, &gMachineAlarms.PERMMEM_FILE_ERROR, gPermData[PERM_CONFIGURATION].IN.PAR.FileName );

					//Make sure the error is acknowledged so we can accept new commands
					gPermData[PERM_CONFIGURATION].IN.CMD.AcknowledgeError = 1;
					CSVFn_Cyclic( &gPermData[PERM_CONFIGURATION] );

					//Append a _tmp so that the file isn't just accepted with invalid values
					strcat(gPermData[PERM_CONFIGURATION].IN.PAR.FileName, "_tmp");

					//Start writing a file and and call cyclicly until it's done
					gPermData[PERM_CONFIGURATION].IN.CMD.SaveVariableListToFile = 1;
					do{
						CSVFn_Cyclic( &gPermData[PERM_CONFIGURATION] );
					}while(	gPermData[PERM_CONFIGURATION].OUT.STAT.Busy  );

					//Call with no commmand to reset for the next file
					gPermData[PERM_CONFIGURATION].IN.CMD.SaveVariableListToFile = 0;
					CSVFn_Cyclic( &gPermData[PERM_CONFIGURATION] );
				}

					//Other errors are just posted to the user and acknowledged to set new files can be created
				else{
					//Alert the user that the config is wrong
					//vfAlarmEdgeSnippet( &gMachineAlarms.components, &gMachineAlarms.PERMMEM_FILE_ERROR, gPermData[PERM_CONFIGURATION].IN.PAR.FileName );

					//Acknowledge the error
					gPermData[PERM_CONFIGURATION].IN.CMD.AcknowledgeError = 1;
					CSVFn_Cyclic( &gPermData[PERM_CONFIGURATION] );
					gPermData[PERM_CONFIGURATION].IN.CMD.AcknowledgeError = 0;
					CSVFn_Cyclic( &gPermData[PERM_CONFIGURATION] );
				}
			} else {
				// no error, mark data valid for this task
				gSplitConfig.taskDataValid[taskIndex] = 1;
			}
		}

		// update datavalid for split config
		gDataValid[PERM_CONFIGURATION] = 1;
		for (taskIndex = 0; taskIndex < gSplitConfig.taskCount; taskIndex++) {
			gDataValid[PERM_CONFIGURATION] &= gSplitConfig.taskDataValid[taskIndex];
		}
	}

	// Initialize non-config persister CSV backups
	strcpy(gPermData[PERM_HOME_DATA].IN.PAR.FileName, "homeData.csv");

	// set non-default gPermData cfg
	gPermData[PERM_HOME_DATA].IN.CFG.MaxFileSize = 10000000;

	for( i = PERM_HOME_DATA; i < NUM_PERSISTERS; i++){

		strcpy(gPermData[i].IN.PAR.FileDevice, "PermData");
		// these array sizes don't inherently match - could cause issues at some point
		memcpy(&gPermData[i].IN.PAR.VariableList, &gPersister[i].IN.WorkingVariableList, sizeof(gPermData[i].IN.PAR.VariableList) );
		strcpy(gPermData[i].IN.CFG.LogFileName, "logs/");
		strcat(gPermData[i].IN.CFG.LogFileName, gPermData[i].IN.PAR.FileName);
		strcat(gPermData[i].IN.CFG.LogFileName, ".log");

		CSVFn_Init(&(gPermData[i]));

		// if persister failed, reload from csv
		if (!gDataValid[i]) {
			CSVOpenFile_Init(&gPermData[i]);
			if (!gPermData[i].OUT.STAT.Error) {
				gDataValid[i] = 1;
			//	vfAlarmEdgeSnippet(&gMachineAlarms.components, &gMachineAlarms.PERMMEM_DATA_RESTORED, gPermData[i].IN.PAR.FileName);
			}
		}

	} // loop through PermData

	// Load configuration.csv every startup
	//CSVOpenFile_Init(&gPermData[PERM_CONFIGURATION]);

} // _INIT
```

#### FirstInitProgCyclic.c - Cyclic code
```c
/********************************************************************
 * COPYRIGHT --
 ********************************************************************
 * Program: FirstInitProg
 * File: FirstInitProgCyclic.c
 * Author: ScismD
 * Created: January 07, 2014
 ********************************************************************
 * Implementation of program FirstInitProg
 ********************************************************************/

#include <bur/plctypes.h>

#ifdef _DEFAULT_INCLUDES
	#include <AsDefault.h>
#endif

void _CYCLIC FirstInitProgCyclic(void)
{
	gCyclic = 1;
	// DO NOT ADD ANY "OTHER" CYCLIC CODE HERE! //
	if( strcmp(_buildDate, gRevInfo_buildDate) != 0 ){
		gTransfer = 1;
	}
}
```

#### FirstInitProg.var - Local variables
```iecst
(********************************************************************
 * COPYRIGHT --
 ********************************************************************
 * Program: FirstInitCProg
 * File: FirstInitCProg.var
 * Author: ScismD
 * Created: January 07, 2014
 ********************************************************************
 * Local variables of program FirstInitCProg
 ********************************************************************)
VAR CONSTANT
	NUM_FILEDEVICES : USINT := 9;
	MAI_FILEDEVICES : USINT := NUM_FILEDEVICES-1;
END_VAR
VAR
	simCheckDevLink : DevLink := (0);
	fileDeviceDevLink : ARRAY[0..MAI_FILEDEVICES] OF DevLink := [9((0))];
	fileDevice : ARRAY[0..MAI_FILEDEVICES] OF STRING[20] := [9('')];
	directory : ARRAY[0..MAI_FILEDEVICES] OF STRING[320] := [9('')];
	parameters : ARRAY[0..MAI_FILEDEVICES] OF STRING[320] := [9('')];
	i : DINT := 0;
	indexString : STRING[320] := '';
	axisString : STRING[320] := '';
	alarmSnippet : STRING[80];
END_VAR
VAR RETAIN
	_buildDate : STRING[80];
END_VAR
```

#### MachineAlarm.var - Local variables
```iecst
VAR
	alarmData : vfAlarms_Data_typ;
	persistErrorID : UINT;
END_VAR
```

### Infrastructure.typ
```iecst
TYPE
	AtnTerminal_typ : 	STRUCT
		Command : STRING[80];
		Console : ARRAY[0..100]OF STRING[80];
		Overflow : ARRAY[0..10]OF STRING[80]; (*:D*)
	END_STRUCT;
	PERM_enum :
		(
		PERM_CONFIGURATION,
		PERM_HOME_DATA,
		PERM_
		);
	SplitConfig_typ : 	STRUCT
		taskDataValid : ARRAY[0..CSV_MAI_VARLIST]OF BOOL;
		taskCount : USINT;
		configList : ARRAY[0..CSV_MAI_VARLIST]OF STRING[PERSIST_STRLEN_VARNAME];
		logFilename : ARRAY[0..CSV_MAI_VARLIST]OF STRING[CSV_STRLEN_FILENAME];
		configFilename : ARRAY[0..CSV_MAI_VARLIST]OF STRING[CSV_STRLEN_FILENAME];
	END_STRUCT;
END_TYPE
```

### Infrastructure.var
```iecst
(*Constants for number of persisters and permanent memory chunks*)
VAR CONSTANT
	NUM_PERSISTERS : USINT := 2;
	MAI_PERSISTERS : USINT := NUM_PERSISTERS-1;
END_VAR
(*Persisters to handle memory management*)
VAR
	gSimulation : BOOL;
	gPersister : ARRAY[0..MAI_PERSISTERS] OF Persistence_typ;
	gPermData : ARRAY[0..MAI_PERSISTERS] OF CSVFileMgr_typ;
END_VAR
VAR RETAIN
	gDataValid : ARRAY[0..MAI_PERSISTERS] OF BOOL;
END_VAR
VAR
	gSplitConfig : SplitConfig_typ;
END_VAR
(*Permanent memory chunks*)
VAR RETAIN
	gPermHomeData : ARRAY[0..MAI_PERM_HOME] OF USINT;
	gPermConfiguration : ARRAY[0..MAI_PERM_CONFIG] OF USINT;
END_VAR
(*ATN*)
VAR CONSTANT
	MAI_PERM_CONFIG : UDINT := 23999;
	MAI_PERM_HOME : UDINT := 1999;
END_VAR
VAR
	gConsole : AtnTerminal_typ;
END_VAR
VAR RETAIN
	gPermDataSize : ARRAY[0..MAI_PERSISTERS] OF UDINT;
END_VAR
VAR
	gCyclic : BOOL;
	gTransfer : BOOL;
	gBootAfterTransfer : BOOL;
END_VAR
```

### Program Logical/Infrastructure/RevInfo/RevInfo (IEC)

#### Main.st
```iecst
PROGRAM _INIT

	gRevInfo_revision;
	revision;	// used for CSVFileMgr headers
	gRevInfo_revisionDate;
	gRevInfo_revisionAuthor;
	gRevInfo_branchName;
	gRevInfo_uncommittedChanges;
	gRevInfo_buildDate;
	gRevInfo_buildConfiguration;
	buildConfiguration;	// used for CSVFileMgr headers
	gRevInfo_builder;
	gRevInfo_versionId;

//	// Create the logger that will be used by RevInfo.
//	createLogInit('App', 1000000, arEVENTLOG_PERSISTENCE_VOLATILE);
//
//	// Log revision information
//	//---------------------------------------------------------------
//
//	logInfo('App', 0, '************ RevInfo Start ************', 0);
//
//	// revision
//	brsmemset(ADR(tempString), 0, SIZEOF(tempString));
//	tempString := 'Revision: ';
//	brsstrcat(ADR(tempString), ADR(revision));
//	logInfo('App', 0, tempString, 0);
//
//	// revisionDate
//	brsmemset(ADR(tempString), 0, SIZEOF(tempString));
//	tempString := 'Commit Date: ';
//	brsstrcat(ADR(tempString), ADR(revisionDate));
//	logInfo('App', 0, tempString, 0);
//
//	// revisionAuthor
//	brsmemset(ADR(tempString), 0, SIZEOF(tempString));
//	tempString := 'Author: ';
//	brsstrcat(ADR(tempString), ADR(revisionAuthor));
//	logInfo('App', 0, tempString, 0);
//
//	// branchName
//	brsmemset(ADR(tempString), 0, SIZEOF(tempString));
//	tempString := 'Branch Name: ';
//	brsstrcat(ADR(tempString), ADR(branchName));
//	logInfo('App', 0, tempString, 0);
//
//	// uncommittedChanges
//	brsmemset(ADR(tempString), 0, SIZEOF(tempString));
//	tempString := 'Uncommitted Changes: ';
//	brsstrcat(ADR(tempString), ADR(uncommittedChanges));
//	logInfo('App', 0, tempString, 0);
//
//	// buildDate
//	brsmemset(ADR(tempString), 0, SIZEOF(tempString));
//	tempString := 'Build Date: ';
//	brsstrcat(ADR(tempString), ADR(buildDate));
//	logInfo('App', 0, tempString, 0);
//
//	// buildConfiguration
//	brsmemset(ADR(tempString), 0, SIZEOF(tempString));
//	tempString := 'Configuration: ';
//	brsstrcat(ADR(tempString), ADR(buildConfiguration));
//	logInfo('App', 0, tempString, 0);
//
//	// builder
//	brsmemset(ADR(tempString), 0, SIZEOF(tempString));
//	tempString := 'Builder: ';
//	brsstrcat(ADR(tempString), ADR(builder));
//	logInfo('App', 0, tempString, 0);
//
//	// versionId
//	brsmemset(ADR(tempString), 0, SIZEOF(tempString));
//	tempString := 'Version ID: ';
//	brsstrcat(ADR(tempString), ADR(versionId));
//	logInfo('App', 0, tempString, 0);
//
//	logInfo('App', 0, '************ RevInfo End ************', 0);

END_PROGRAM
```

- getRevInfo.sh (not shown)

### RevInfo.var
```iecst
(* RevInfo.var 2.0.0 *)
VAR CONSTANT
	gRevInfo_revision : STRING[80] := '8d98d94';
	revision : STRING[80] := '8d98d94';
	gRevInfo_revisionDate : STRING[80] := '2025-09-05 16:52:17 -0400';
	gRevInfo_revisionAuthor : STRING[80] := 'Harshith';
	gRevInfo_branchName : STRING[80] := 'main';
	gRevInfo_uncommittedChanges : STRING[80] := ' 11061 files changed, 46 insertions(+), 2516071 deletions(-)';
	gRevInfo_buildDate  : STRING[80] := '2025-09-08 11:38:32 -0400';
	gRevInfo_buildConfiguration : STRING[80] := 'ControlPLC_DataDistribution';
	buildConfiguration : STRING[80] := 'ControlPLC_DataDistribution';
	gRevInfo_builder : STRING[80] := 'hkeshavamurthy';
	gRevInfo_versionId : STRING[80] := '8d98d94';
END_VAR
```

### Program Logical/Infrastructure/atnDriver (IEC)

#### Variables.var
```iecst
VAR
	execute : BOOL;
END_VAR
```

#### Main.st
```iecst
PROGRAM _CYCLIC

	atncyclic( ADR(gConsole.Command), SIZEOF(gConsole.Command) );

END_PROGRAM
```

### Alarms.typ
```iecst
TYPE
	AlarmApi : 	STRUCT
		cores : STRING[80];
	END_STRUCT;
END_TYPE
```

### Alarms.var
```iecst
VAR
	gAlarmApi : AlarmApi;
END_VAR
```

### Program Logical/Infrastructure/Alarms/AlarmWrap (IEC)

#### Types.typ
```iecst
TYPE
	IO_DI_typ : 	STRUCT
		operatorStationAckAll : BOOL;
	END_STRUCT;
	IO_DO_typ : 	STRUCT
		operatorStationAlarmsLED : BOOL;
	END_STRUCT;
	IO_typ : 	STRUCT
		di : IO_DI_typ;
		do : IO_DO_typ;
	END_STRUCT;
END_TYPE
```

#### Variables.var
```iecst
VAR
	wrapper : {REDUND_UNREPLICABLE} errWrap_typ;
	selectedIndex : UDINT;
	selectedName : STRING[80];
	prevSelectedIndex : UDINT;
	activeAlarmSeverity : ARRAY[0..ERRWRAP_MAI_ERRORS_DISP] OF STRING[20];
	i : INT;
	dAlarmComponent : REFERENCE TO vfAlarms_Component_typ;
	pAlarmComponent : {REDUND_UNREPLICABLE} UDINT;
	sAlarmComponent : {REDUND_UNREPLICABLE} UDINT;
	newLink : {REDUND_UNREPLICABLE} MpComIdentType;
	coreNames : ARRAY[0..25] OF STRING[80];
	coreAlarmsPresent : ARRAY[0..25] OF BOOL;
	oldLink : MpComIdentType;
	IO : IO_typ;
	_operatorStationAckAll : BOOL;
	blinkLED : Blink;
	displayAble : INT;
	snippet : STRING[80];
	dSelectedAlarmCore : REFERENCE TO MpAlarmXCore;
END_VAR
```

#### Main.st
```iecst
PROGRAM _INIT

	// Set defaults
	wrapper.internal.mpAlarmX := ADR(gMachineAlarms.components.core);
	wrapper.in.par.coreMpLink := ADR(gMachineAlarms.components.link);

	//Init alarm wrapper
	//	//Configure History FUB
	//	wrapper.in.par.histMpLink := ADR(gAlarmXHistory_Machine);
	//	wrapper.internal.mpAlarmXHistory.Enable := TRUE;
	//	wrapper.internal.mpAlarmXHistory.MpLink := wrapper.in.par.histMpLink;

	//Configure Core List UI
	wrapper.in.par.uiCoreSetup.AlarmListSize := 30;
	wrapper.internal.mpAlarmXListUI.Enable := TRUE;
	wrapper.internal.mpAlarmXListUI.UIConnect := ADR(wrapper.internal.uiCoreConnect);
	wrapper.internal.mpAlarmXListUI.MpLink := wrapper.in.par.coreMpLink;
	wrapper.internal.mpAlarmXListUI.UISetup := wrapper.in.par.uiCoreSetup;

	//	//Configure History List UI
	//	wrapper.internal.mpAlarmXHistoryUI.Enable := TRUE;
	//	wrapper.internal.mpAlarmXHistoryUI.UIConnect := ADR(wrapper.internal.uiHistConnect);
	//	wrapper.internal.mpAlarmXHistoryUI.MpLink := wrapper.in.par.histMpLink;
	//	wrapper.internal.mpAlarmXHistoryUI.UISetup := wrapper.in.par.uiHistSetup;

	//Configure Acknowledge all FUB
	wrapper.internal.mpAcknowledgeAll.Enable := 1;
	wrapper.internal.mpAcknowledgeAll.MpLink := wrapper.in.par.coreMpLink;
	wrapper.internal.uiCoreConnect.AcknowledgeAll := 1; //acknowledge on boot

	wrapper.in.cfg.errorSeverity; 	// Not used
	wrapper.in.cfg.logSeverity; 	// Not used

	blinkLED.Enable := TRUE;
	blinkLED.Time := T#2s;
	blinkLED.Percentage := 50;

END_PROGRAM

PROGRAM _CYCLIC

	displayAble := 0;
	// call all alarm cores
	FOR i:=0 TO stateCount(gAlarmApi.cores) BY 1 DO
		IF forStateGetPointer(gAlarmApi.cores, i, 0, ADR(pAlarmComponent), ADR(sAlarmComponent)) THEN
			dAlarmComponent ACCESS pAlarmComponent;
			dAlarmComponent.core.Enable := TRUE;
			dAlarmComponent.core.MpLink := ADR(dAlarmComponent.link);
			dAlarmComponent.core();
			//dAlarmComponent.core.ErrorReset := dAlarmComponent.core.Error;

			IF NOT dAlarmComponent.noDisplay THEN
				IF displayAble = selectedIndex THEN
					newLink := dAlarmComponent.link;
					wrapper.internal.mpAlarmX := ADR(dAlarmComponent.core);
					selectedName := dAlarmComponent.name;
				END_IF

				coreNames[displayAble] := dAlarmComponent.name;
				coreNames[displayAble] := CONCAT(coreNames[displayAble], ' (');

				coreNames[displayAble] := CONCAT(coreNames[displayAble], ' Active: ');
				brsitoa(dAlarmComponent.core.ActiveAlarms, ADR(snippet));
				coreNames[displayAble] := CONCAT(coreNames[displayAble], snippet);

				coreNames[displayAble] := CONCAT(coreNames[displayAble], ' Pending: ');
				brsitoa(dAlarmComponent.core.PendingAlarms, ADR(snippet));
				coreNames[displayAble] := CONCAT(coreNames[displayAble], snippet);

				coreNames[displayAble] := CONCAT(coreNames[displayAble], ' )');

				IF ((dAlarmComponent.core.ActiveAlarms > 0) OR (dAlarmComponent.core.PendingAlarms > 0)) THEN
					coreAlarmsPresent[displayAble] := TRUE;
				ELSE
					coreAlarmsPresent[displayAble] := FALSE;
				END_IF

				displayAble := displayAble + 1;
			END_IF
		END_IF
	END_FOR

	IF oldLink.Internal[0] <> newLink.Internal[0] THEN

		oldLink := newLink;

		// disable
		//		wrapper.internal.mpAlarmX.Enable := FALSE;
		wrapper.internal.mpAcknowledgeAll.Enable := FALSE;
		wrapper.internal.mpAlarmXListUI.Enable := FALSE;
		errorWrapCyclic(wrapper);

		// reenable with new selection
		//		wrapper.internal.mpAlarmX.Enable := TRUE;
		wrapper.internal.mpAcknowledgeAll.Enable := TRUE;
		wrapper.internal.mpAlarmXListUI.Enable := TRUE;

	END_IF

	// Map the operator station command to acknowledge all alarms.
	IF (IO.di.operatorStationAckAll AND NOT _operatorStationAckAll) THEN
		_operatorStationAckAll := TRUE;
		wrapper.in.cmd.acknowledgeAllAlarms := TRUE;
	ELSIF (NOT IO.di.operatorStationAckAll) THEN
		_operatorStationAckAll := FALSE;
	END_IF
	// Map the operator station alarm indicator to the presence of alarms.
	// It should be solid if acknowledged alarms are present,
	// and blink if unacknowledged alarms are present.
	IF (wrapper.out.alarmPresent) THEN
		// TODO: check if alarms are ack'd, and change to solid.
		IO.do.operatorStationAlarmsLED := blinkLED.Out;
	END_IF
	blinkLED();

	wrapper.in.par.coreMpLink := ADR(newLink);
	//	wrapper.internal.mpAlarmX.MpLink := wrapper.in.par.coreMpLink;
	wrapper.internal.mpAcknowledgeAll.MpLink := wrapper.in.par.coreMpLink;
	wrapper.internal.mpAlarmXListUI.MpLink := wrapper.in.par.coreMpLink;
	errorWrapCyclic(wrapper);

	// Use a dynamic variable for watch window access
	dSelectedAlarmCore ACCESS wrapper.internal.mpAlarmX;

	FOR i := 0 TO ERRWRAP_MAI_ERRORS_DISP BY 1 DO
		IF wrapper.out.activeAlarmInfo[i].code <> 0 THEN
			wrapper.out.activeAlarmInfo[i].codeString := UDINT_TO_STRING(wrapper.out.activeAlarmInfo[i].code);
		ELSE
			wrapper.out.activeAlarmInfo[i].codeString := '';
		END_IF
		CASE wrapper.out.activeAlarmInfo[i].severity OF

			vfALARMS_SEVERITY_NONE:
				activeAlarmSeverity[i] := '';

			vfALARMS_SEVERITY_INFO:
				activeAlarmSeverity[i] := 'INFO';

			vfALARMS_SEVERITY_WARNING:
				activeAlarmSeverity[i] := 'WARN';

			vfALARMS_SEVERITY_ALARM:
				activeAlarmSeverity[i] := 'STOP';

			vfALARMS_SEVERITY_CRITICAL:
				activeAlarmSeverity[i] := 'ABORT';

		END_CASE
	END_FOR

END_PROGRAM

PROGRAM _EXIT

END_PROGRAM
```

### Package Logical/Libraries - Global libraries

### Library Logical/Libraries/Loupe/errorAPI (ANSIC)
Depends on: AsBrStr, MpAlarmX

#### Types.typ - Exported data types
```iecst
TYPE
	errWrap_typ : 	STRUCT
		in : errWrapIn_typ;
		out : errWrapOut_typ;
		internal : errWrapInternal_typ;
	END_STRUCT;
	errWrapIn_typ : 	STRUCT
		cmd : errWrapInCmd_typ;
		par : errWrapInPar_typ;
		cfg : errWrapInCfg_typ;
	END_STRUCT;
	errWrapInCmd_typ : 	STRUCT
		acknowledgeError : BOOL;
		acknowledgeAllAlarms : BOOL;
		exportHistory : BOOL;
	END_STRUCT;
	errWrapInPar_typ : 	STRUCT
		coreMpLink : REFERENCE TO MpComIdentType;
		histMpLink : REFERENCE TO MpComIdentType;
		uiHistSetup : MpAlarmXHistoryUISetupType;
		uiCoreSetup : MpAlarmXListUISetupType;
	END_STRUCT;
	errWrapInCfg_typ : 	STRUCT
		logSeverity : UDINT;
		errorSeverity : UDINT;
	END_STRUCT;
	errWrapAlarmOut_typ : 	STRUCT
		scope : STRING[255];
		name : STRING[255];
		message : STRING[255];
		additionalInfo : STRING[255];
		code : UDINT;
		instance : UDINT;
		severity : UDINT;
		timeStamp : STRING[50];
		codeString : STRING[7];
	END_STRUCT;
	errWrapOut_typ : 	STRUCT
		activeAlarms : UINT;
		error : BOOL;
		errorID : UINT;
		errorString : STRING[320];
		activeAlarmInfo : ARRAY[0..ERRWRAP_MAI_ERRORS_DISP]OF errWrapAlarmOut_typ;
		alarmPresent : BOOL;
		wStrMessage : ARRAY[0..ERRWRAP_MAI_ERRORS_DISP]OF WSTRING[255];
		wStrAdditionalInfo : ARRAY[0..ERRWRAP_MAI_ERRORS_DISP]OF WSTRING[255];
	END_STRUCT;
	errWrapInternal_typ : 	STRUCT
		userAlarms : ARRAY[0..ERRWRAP_MAI_ERRORS]OF errWrapInternalAlarm_typ;
		activeAlarms : UINT;
		initialized : BOOL;
		id : UDINT;
		coreMpLink : REFERENCE TO MpComIdentType;
		histMpLink : MpComIdentType;
		exportHistory : BOOL;
		resetErrors : BOOL;
		mpAlarmX : REFERENCE TO MpAlarmXCore;
		mpAlarmXHistory : MpAlarmXHistory;
		mpAlarmXListUI : MpAlarmXListUI;
		mpAlarmXHistoryUI : MpAlarmXHistoryUI;
		resetErrorCounter : USINT;
		resetCounter : USINT;
		uiHistConnect : MpAlarmXHistoryUIConnectType;
		uiCoreConnect : MpAlarmXListUIConnectType;
		mpAcknowledgeAll : MpAlarmXAcknowledgeAll;
		previousActiveCount : UINT;
		alarmListLoopIndex : USINT;
		alarmListActiveCount : USINT;
		_previousAlarmMessage : STRING[255];
		_previousAlarmMessageList : ARRAY[0..ERRWRAP_MAI_ERRORS_DISP]OF STRING[255];
		_previousAlarmListActiveCount : USINT;
		_previousWrapperAlarmActiveCount : USINT;
	END_STRUCT;
	errWrapInternalAlarm_typ : 	STRUCT
		name : STRING[80];
		active : BOOL;
		set : BOOL;
		id : UDINT;
		configure : MpAlarmXConfigAlarm;
		behavoir : MpAlarmXAlarmConfigType;
		acknowledge : UDINT;
		timeStamp : DATE_AND_TIME;
	END_STRUCT;
	alarmX_ST_enum :
		(
		ALARMX_IDLE_ST,
		ALARMX_EXPORT_HISTORY_ST,
		ALARMX_RESET_FUBS_ST,
		ALARMX_ACK_ALL_ST,
		ALARMX_RESET_ALARMS_ST
		);
END_TYPE
```

#### Constants.var - Exported constants
```iecst
VAR CONSTANT
	ERRWRAP_NUM_ERRORS : USINT := 50;
	ERRWRAP_MAI_ERRORS : USINT := ERRWRAP_NUM_ERRORS-1;
	ERRWRAP_NUM_ERRORS_DISP : USINT := 30;
	ERRWRAP_MAI_ERRORS_DISP : USINT := ERRWRAP_NUM_ERRORS_DISP-1;
END_VAR
```

#### errorAPI.fun - Exported functions and function blocks
```iecst
FUNCTION errorWrapCyclic : USINT
	VAR_INPUT
		inst : errWrap_typ;
	END_VAR
END_FUNCTION

FUNCTION errorWrapAck : UDINT
	VAR_INPUT
		id : UDINT;
		alarmCollector : errWrap_typ;
	END_VAR
END_FUNCTION

FUNCTION errorWrapSet : UDINT
	VAR_INPUT
		source : UDINT;
		string : UDINT;
		errorId : UDINT;
		acknowledge : UDINT;
		alarmCollector : errWrap_typ;
	END_VAR
END_FUNCTION
```

#### cyclic.c
```c
#include <bur/plctypes.h>
#ifdef __cplusplus
	extern "C"
	{
#endif

#include "errorAPI.h"

#ifdef __cplusplus
	};
#endif

#include "string.h"

unsigned char errorWrapCyclic(errWrap_typ* inst) {
	int i;
	int numMappAlarms;
	int outputIndex;
	int mpAlarmIndex;

	if (inst->in.cmd.acknowledgeAllAlarms){
		inst->in.cmd.acknowledgeAllAlarms = 0;
		inst->internal.mpAcknowledgeAll.Execute = 1;
		brsmemset(&inst->out.activeAlarmInfo, 0, sizeof(inst->out.activeAlarmInfo));
	}
	else{
		inst->internal.mpAcknowledgeAll.Execute = 0;
	}

	//Cyclically call FUBs
//	MpAlarmXCore(inst->internal.mpAlarmX);	// call each core in the wrapper task because we need many cores
	MpAlarmXHistory(&inst->internal.mpAlarmXHistory);
	MpAlarmXListUI(&inst->internal.mpAlarmXListUI);
	MpAlarmXHistoryUI(&inst->internal.mpAlarmXHistoryUI);
	MpAlarmXAcknowledgeAll(&inst->internal.mpAcknowledgeAll);

	if(!inst->internal.initialized) {
		char tempString[10];
		inst->internal.initialized = 1;
		for (i = 0; i < ERRWRAP_NUM_ERRORS; i++) {
			brsitoa(i, tempString);
			strcpy(inst->internal.userAlarms[i].name, "TempAlarm");
			strcat(inst->internal.userAlarms[i].name, tempString);

			inst->internal.userAlarms[i].configure.MpLink = inst->in.par.coreMpLink;
			inst->internal.userAlarms[i].configure.Name = &inst->internal.userAlarms[i].name;
			inst->internal.userAlarms[i].configure.Configuration = &inst->internal.userAlarms[i].behavoir;
			inst->internal.userAlarms[i].behavoir.Behavior.AutoReset = 1;
			inst->internal.userAlarms[i].behavoir.Behavior.Acknowledge = mpALARMX_ACK_REQ;
			inst->internal.userAlarms[i].configure.Enable = 1;
			//inst->internal.alarms[i].behavoir.Severity
		}
	}

	inst->internal.activeAlarms = 0; // ReCount active errors cyclically
	for (i = 0; i < ERRWRAP_NUM_ERRORS; i++) {

		if(inst->internal.userAlarms[i].active) {
			inst->internal.activeAlarms++;
		}

		MpAlarmXConfigAlarm(&inst->internal.userAlarms[i].configure);

		if(inst->internal.userAlarms[i].active &&
			inst->internal.userAlarms[i].configure.Active
		&& !inst->internal.userAlarms[i].set) {
			inst->internal.userAlarms[i].configure.Save = 1;
		}

		if(inst->internal.userAlarms[i].configure.Save && inst->internal.userAlarms[i].configure.CommandDone){
			inst->internal.userAlarms[i].set = 1;
			inst->internal.userAlarms[i].configure.Save = 0;
			MpAlarmXSet(inst->internal.userAlarms[i].configure.MpLink, inst->internal.userAlarms[i].name);
		}

		if(inst->internal.userAlarms[i].set) {
			if(MpAlarmXCheckState(inst->internal.userAlarms[i].configure.MpLink, inst->internal.userAlarms[i].name, mpALARMX_STATE_NONE)) {
				// Alarm was acknowledged and reset (reset is automatic)
				inst->internal.userAlarms[i].set = 0;
				inst->internal.userAlarms[i].active = 0;

				if(inst->internal.userAlarms[i].acknowledge) {
					*((BOOL*)inst->internal.userAlarms[i].acknowledge) = 1;
				}
			}
		}

	}

	// Set outputs

	outputIndex = 0;

	for (i = 0; i < ERRWRAP_NUM_ERRORS_DISP; i++){
		brsmemcpy(&inst->out.activeAlarmInfo[outputIndex].name, &inst->internal.uiCoreConnect.AlarmList.Name[i], sizeof(inst->out.activeAlarmInfo[outputIndex].name));
		brsmemcpy(&inst->out.activeAlarmInfo[outputIndex].scope, &inst->internal.uiCoreConnect.AlarmList.Scope[i], sizeof(inst->out.activeAlarmInfo[outputIndex].scope));
		brsmemcpy(&inst->out.wStrMessage[outputIndex], &inst->internal.uiCoreConnect.AlarmList.Message[i], sizeof(inst->out.wStrMessage[outputIndex]));
		brsmemcpy(&inst->out.wStrAdditionalInfo[outputIndex], &inst->internal.uiCoreConnect.AlarmList.AdditionalInformation1[i], sizeof(inst->out.wStrAdditionalInfo[outputIndex]));
		brsstrcpy((UDINT)&inst->out.activeAlarmInfo[outputIndex].timeStamp,(UDINT)&inst->internal.uiCoreConnect.AlarmList.Timestamp[i]);
		inst->out.activeAlarmInfo[outputIndex].severity = inst->internal.uiCoreConnect.AlarmList.Severity[i];
		inst->out.activeAlarmInfo[outputIndex].code = inst->internal.uiCoreConnect.AlarmList.Code[i];
		inst->out.activeAlarmInfo[outputIndex].instance = inst->internal.uiCoreConnect.AlarmList.InstanceID[i];
		wstring2string( &inst->out.activeAlarmInfo[outputIndex].message, &inst->out.wStrMessage[outputIndex], sizeof(inst->out.activeAlarmInfo[outputIndex].message) );
		wstring2string( &inst->out.activeAlarmInfo[outputIndex].additionalInfo, &inst->out.wStrAdditionalInfo[outputIndex], sizeof(inst->out.activeAlarmInfo[outputIndex].additionalInfo) );
		outputIndex++;
	}

	if(inst->out.activeAlarms > 0){
		inst->out.alarmPresent = 1;
	}
	else{
		inst->out.alarmPresent = 0;
	}

	inst->out.activeAlarms = inst->internal.mpAlarmX->PendingAlarms + inst->internal.mpAlarmX->ActiveAlarms;
		return 0;
}
```

#### setAlarm.c
```c
#include <bur/plctypes.h>
#ifdef __cplusplus
	extern "C"
	{
#endif

#include "errorAPI.h"

#ifdef __cplusplus
	};
#endif

#include "string.h"

unsigned long errorWrapSet(unsigned long source, unsigned long string, unsigned long errorId, unsigned long acknowledge, struct errWrap_typ* alarmCollector) {
	UINT i;

	if(alarmCollector == 0) return 1;

	alarmCollector->internal.id++; // Make sure every alarm has a unique id

	for (i = 0; i < ERRWRAP_NUM_ERRORS; i++) {
		if(!alarmCollector->internal.userAlarms[i].active) {
			alarmCollector->internal.userAlarms[i].active = 1;
			alarmCollector->internal.userAlarms[i].configure.Enable = 1;
			alarmCollector->internal.userAlarms[i].id = alarmCollector->internal.id;

			alarmCollector->internal.userAlarms[i].behavoir.Code = errorId;

			// Set message
			alarmCollector->internal.userAlarms[i].behavoir.Message[0] = '\0';
			if(source) {
				strcat(alarmCollector->internal.userAlarms[i].behavoir.Message, source);
				strcat(alarmCollector->internal.userAlarms[i].behavoir.Message, ": ");
			}
			if(string) {
				strcat(alarmCollector->internal.userAlarms[i].behavoir.Message, string);
			}

			alarmCollector->internal.userAlarms[i].acknowledge = acknowledge;

			break;
		}
	}

	return 0;
}
```

#### ackAlarm.c
```c
#include <bur/plctypes.h>
#ifdef __cplusplus
	extern "C"
	{
#endif

#include "errorAPI.h"

#ifdef __cplusplus
	};
#endif

#include "string.h"

unsigned long errorWrapAck(unsigned long id, struct errWrap_typ* alarmCollector) {
	UINT i;

	if(alarmCollector == 0) return 1;

	for (i = 0; i < ERRWRAP_NUM_ERRORS; i++) {
		if(alarmCollector->internal.userAlarms[i].id == id) {
			if(alarmCollector->internal.userAlarms[i].active) {
				alarmCollector->internal.userAlarms[i].active = 0;
				alarmCollector->internal.userAlarms[i].set = 0;

				if(alarmCollector->internal.userAlarms[i].set) {
					// Ack
					MpAlarmXAcknowledge(alarmCollector->internal.userAlarms[i].configure.MpLink, alarmCollector->internal.userAlarms[i].name);
				}
				else {
					// Stop configuring
					alarmCollector->internal.userAlarms[i].configure.Enable = 0;
					// Call this so if we can use this index again before running the cylic
					MpAlarmXConfigAlarm(&alarmCollector->internal.userAlarms[i].configure);
				}
			}
			break;
		}
	}

	return 0;
}
```

### Library Logical/Libraries/VF/VFAlarms (ANSIC, version 0.01.0)
Depends on: MpCom, AsXml, fiowrap, AsBrStr, MpAlarmX

#### Types.typ - Exported data types
```iecst
TYPE
	vfAlarms_Data_typ : 	STRUCT
		in : vfAlarms_Data_In_typ;
		out : vfAlarms_Data_Out_typ;
		internal : vfAlarms_Data_Internal_typ;
	END_STRUCT;
	vfAlarms_Data_In_typ : 	STRUCT
		mpLink : UDINT;
		deviceName : STRING[80];
		scope : STRING[80];
		mpLinkName : STRING[80];
		snippetPvName : STRING[80];
		escalateAll : BOOL;
	END_STRUCT;
	vfAlarms_Data_Internal_typ : 	STRUCT
		fub : vfAlarms_Data_Internal_Fub_typ;
		defaultMapping : vfAlarms_DefaultMapping_typ;
		alarms : ARRAY[0..vfALARMS_MAI_ALARMS]OF vfAlarms_Item_typ;
		snippets : ARRAY[0..vfALARMS_MAI_SNIPPETS]OF vfAlarms_Snippet_typ;
		reactions : vfAlarms_Reactions_typ;
		aggregations : vfAlarms_Aggregations_typ;
		fileName : STRING[80];
		xmlIdent : UDINT;
		pXmlData : UDINT;
		szXmlData : UDINT;
	END_STRUCT;
	vfAlarms_DefaultMapping_typ : 	STRUCT
		type : vfALARMS_MAPPING_enum;
		alarmName : STRING[vfALARMS_MAX_NAME_LEN];
	END_STRUCT;
	vfAlarms_Aggregations_typ : 	STRUCT
		byName : ARRAY[0..vfALARMS_MAI_MAPPINGS]OF vfAlarms_AggByName_typ;
		bySeverity : ARRAY[0..vfALARMS_MAI_MAPPINGS]OF vfAlarms_AggBySeverity_typ;
	END_STRUCT;
	vfAlarms_AggByName_typ : 	STRUCT
		name : STRING[vfALARMS_MAX_NAME_LEN];
		aggregationName : STRING[vfALARMS_MAX_NAME_LEN];
	END_STRUCT;
	vfAlarms_AggBySeverity_typ : 	STRUCT
		severity : vfALARMS_SEVERITY_enum;
		aggregationName : STRING[vfALARMS_MAX_NAME_LEN];
	END_STRUCT;
	vfAlarms_Reactions_typ : 	STRUCT
		byNameNotEscalated : ARRAY[0..vfALARMS_MAI_MAPPINGS]OF vfAlarms_ReactionByName_typ;
		byName : ARRAY[0..vfALARMS_MAI_MAPPINGS]OF vfAlarms_ReactionByName_typ;
		bySeverity : ARRAY[0..vfALARMS_MAI_MAPPINGS]OF vfAlarms_ReactionBySeverity_typ;
	END_STRUCT;
	vfAlarms_ReactionByName_typ : 	STRUCT
		name : STRING[vfALARMS_MAX_NAME_LEN];
		reactionName : ARRAY[0..vfALARMS_MAI_REACTIONS]OF STRING[vfALARMS_MAX_REACTION_LEN];
	END_STRUCT;
	vfAlarms_ReactionBySeverity_typ : 	STRUCT
		severity : vfALARMS_SEVERITY_enum;
		reactionName : ARRAY[0..vfALARMS_MAI_REACTIONS]OF STRING[vfALARMS_MAX_REACTION_LEN];
	END_STRUCT;
	vfAlarms_Data_Internal_Fub_typ : 	STRUCT
		manageConfiguration : MpComConfigManager;
		xmlCreateMemoryWriter : xmlCreateMemoryWriter;
		xmlWriteStartDocument : xmlWriteStartDocument;
		xmlWriteStartElement : xmlWriteStartElement;
		xmlWriteAttribute : xmlWriteAttribute;
		xmlWriteEndElement : xmlWriteEndElement;
		xmlWriteEndDocument : xmlWriteEndDocument;
		xmlGetMemoryInfo : xmlGetMemoryInfo;
		xmlCloseMemoryWriter : xmlCloseMemoryWriter;
		fioWrapper : FIOWrap_typ;
	END_STRUCT;
	vfAlarms_Data_Out_typ : 	STRUCT
		done : BOOL;
		error : BOOL;
		errorId : DINT;
		errorString : STRING[80];
	END_STRUCT;
	vfAlarms_Item_typ : 	STRUCT
		name : STRING[vfALARMS_MAX_NAME_LEN];
		scope : STRING[vfALARMS_MAX_NAME_LEN];
		textScope : STRING[vfALARMS_MAX_NAME_LEN];
		code : UDINT;
		severity : vfALARMS_SEVERITY_enum;
		behavior : vfALARMS_BEHAVIOR_enum;
	END_STRUCT;
	vfAlarms_Snippet_typ : 	STRUCT
		key : STRING[vfALARMS_MAX_SNIPPET_KEY_LEN];
		pvName : STRING[vfALARMS_MAX_SNIPPET_PV_NAME_LEN];
	END_STRUCT;
	vfAlarms_Component_typ : 	STRUCT
		link : {REDUND_UNREPLICABLE} MpComIdentType;
		core : {REDUND_UNREPLICABLE} MpAlarmXCore;
		noDisplay : BOOL;
		name : STRING[80];
	END_STRUCT;
	vfAlarms_Instance_type : 	STRUCT
		_ : STRING[80];
		id : UDINT;
		snippet : STRING[vfALARMS_MAX_SNIPPET_STR_LENGTH];
	END_STRUCT;
	Log_Origin_Mappings_typ : 	STRUCT
		originFormatted : ARRAY[0..LOGBOOK_MAI_MAPPINGS]OF STRING[32];
		originRaw : ARRAY[0..LOGBOOK_MAI_MAPPINGS]OF STRING[32];
	END_STRUCT;
	vfALARMS_MAPPING_enum :
		(
		vfALARMS_MAPPING_REMAIN,
		vfALARMS_MAPPING_AGGREGATE,
		vfALARMS_MAPPING_ESCALATE
		);
	vfALARMS_BEHAVIOR_enum :
		(
		vfALARMS_BEHAVIOR_PERSISTENT,
		vfALARMS_BEHAVIOR_EDGE
		);
	vfALARMS_SEVERITY_enum :
		(
		vfALARMS_SEVERITY_NONE := 0,
		vfALARMS_SEVERITY_INFO := 1,
		vfALARMS_SEVERITY_WARNING := 2,
		vfALARMS_SEVERITY_ALARM := 3,
		vfALARMS_SEVERITY_CRITICAL := 4
		);
	vfALARMS_XML_TYPE_enum :
		(
		vfALARMS_XML_TYPE_START_WRITE,
		vfALARMS_XML_TYPE_START_DOC,
		vfALARMS_XML_TYPE_START_ELEM,
		vfALARMS_XML_TYPE_ATTRIBUTE,
		vfALARMS_XML_TYPE_END_ELEM,
		vfALARMS_XML_TYPE_END_DOC,
		vfALARMS_XML_TYPE_GET_MEM,
		vfALARMS_XML_TYPE_END_WRITE
		);
	vfALARMS_FILE_CMD_enum :
		(
		vfALARMS_FILE_CMD_DELETE,
		vfALARMS_FILE_CMD_SAVE
		);
END_TYPE
```

#### Constants.var - Exported constants
```iecst
VAR CONSTANT
	vfALARMS_MAX_NAME_LEN : UINT := 80;
	vfALARMS_MAX_REACTION_LEN : UINT := 80;
	vfALARMS_MAX_BEHAVIOR_LEN : UINT := 80;
	vfALARMS_MAX_SNIPPET_KEY_LEN : UINT := 80;
	vfALARMS_MAX_SNIPPET_PV_NAME_LEN : UINT := 80;
	vfALARMS_MAX_SNIPPET_STR_LENGTH : UINT := 255;
	vfALARMS_MAX_ALARMS : UINT := 100;
	vfALARMS_MAI_ALARMS : UINT := vfALARMS_MAX_ALARMS-1;
	vfALARMS_MAX_SNIPPETS : UINT := 100;
	vfALARMS_MAI_SNIPPETS : UINT := vfALARMS_MAX_SNIPPETS-1;
	vfALARMS_MAX_MAPPINGS : UINT := 100;
	vfALARMS_MAI_MAPPINGS : UINT := vfALARMS_MAX_MAPPINGS-1;
	vfALARMS_MAX_REACTIONS : UINT := 6;
	vfALARMS_MAI_REACTIONS : UINT := vfALARMS_MAX_REACTIONS-1;
	vfALARMS_MAX_BUFFER_LEN : UDINT := 1500000;
	vfALARMS_MAI_BUFFER : UDINT := vfALARMS_MAX_BUFFER_LEN-1;
	LOGBOOK_MAI_MAPPINGS : UINT := 200;
END_VAR
```

#### VFAlarms.fun - Exported functions and function blocks
```iecst
{REDUND_ERROR} FUNCTION vfAddSnippet : BOOL (* *) (*$GROUP=User,$CAT=User,$GROUPICON=User.png,$CATICON=User.png*)
	VAR_INPUT
		key : STRING[vfALARMS_MAX_SNIPPET_KEY_LEN]; (*The name of the snippet that will be referenced in a TMX file (i.e. via {&snippet})*)
		pvName : STRING[vfALARMS_MAX_SNIPPET_PV_NAME_LEN]; (*The name of the PV, including task name (i.e. ::myTask:MyPV)*)
	END_VAR
	VAR_IN_OUT
		data : vfAlarms_Data_typ; (*The VfAlarms data structure that stores transient info*)
	END_VAR
END_FUNCTION

{REDUND_ERROR} FUNCTION vfAddAggregationBySeverity : BOOL (* *) (*$GROUP=User,$CAT=User,$GROUPICON=User.png,$CATICON=User.png*)
	VAR_INPUT
		severity : vfALARMS_SEVERITY_enum; (*The severity that triggers this aggregation*)
		aggregationName : STRING[vfALARMS_MAX_NAME_LEN]; (*The name of the alarm that gets escalated during aggregation*)
	END_VAR
	VAR_IN_OUT
		data : vfAlarms_Data_typ; (*The VfAlarms data structure that stores transient info*)
	END_VAR
END_FUNCTION

{REDUND_ERROR} FUNCTION vfAddAggregationByName : BOOL (* *) (*$GROUP=User,$CAT=User,$GROUPICON=User.png,$CATICON=User.png*)
	VAR_INPUT
		name : STRING[vfALARMS_MAX_NAME_LEN]; (*The alarm name that triggers the aggregation*)
		aggregationName : STRING[vfALARMS_MAX_NAME_LEN]; (*The name of the alarm that gets escalated during aggregation*)
	END_VAR
	VAR_IN_OUT
		data : vfAlarms_Data_typ; (*The VfAlarms data structure that stores transient info*)
	END_VAR
END_FUNCTION

{REDUND_ERROR} FUNCTION vfAddReactionBySeverity : BOOL (* *) (*$GROUP=User,$CAT=User,$GROUPICON=User.png,$CATICON=User.png*)
	VAR_INPUT
		severity : vfALARMS_SEVERITY_enum; (*The severity that triggers these reactions*)
		reactionName1 : STRING[vfALARMS_MAX_REACTION_LEN]; (*A reaction that gets triggered by the associated severity*)
		reactionName2 : STRING[vfALARMS_MAX_REACTION_LEN]; (*A reaction that gets triggered by the associated severity*)
		reactionName3 : STRING[vfALARMS_MAX_REACTION_LEN]; (*A reaction that gets triggered by the associated severity*)
		reactionName4 : STRING[vfALARMS_MAX_REACTION_LEN]; (*A reaction that gets triggered by the associated severity*)
		reactionName5 : STRING[vfALARMS_MAX_REACTION_LEN]; (*A reaction that gets triggered by the associated severity*)
		reactionName6 : STRING[vfALARMS_MAX_REACTION_LEN]; (*A reaction that gets triggered by the associated severity*)
	END_VAR
	VAR_IN_OUT
		data : vfAlarms_Data_typ; (*The VfAlarms data structure that stores transient info*)
	END_VAR
END_FUNCTION

{REDUND_ERROR} FUNCTION vfAddReactionByName : BOOL (* *) (*$GROUP=User,$CAT=User,$GROUPICON=User.png,$CATICON=User.png*)
	VAR_INPUT
		name : STRING[vfALARMS_MAX_NAME_LEN]; (*The alarm name that triggers these reactions*)
		reactionName1 : STRING[vfALARMS_MAX_REACTION_LEN]; (*A reaction that gets triggered by the associated alarm name*)
		reactionName2 : STRING[vfALARMS_MAX_REACTION_LEN]; (*A reaction that gets triggered by the associated alarm name*)
		reactionName3 : STRING[vfALARMS_MAX_REACTION_LEN]; (*A reaction that gets triggered by the associated alarm name*)
		reactionName4 : STRING[vfALARMS_MAX_REACTION_LEN]; (*A reaction that gets triggered by the associated alarm name*)
		reactionName5 : STRING[vfALARMS_MAX_REACTION_LEN]; (*A reaction that gets triggered by the associated alarm name*)
		reactionName6 : STRING[vfALARMS_MAX_REACTION_LEN]; (*A reaction that gets triggered by the associated alarm name*)
	END_VAR
	VAR_IN_OUT
		data : vfAlarms_Data_typ; (*The VfAlarms data structure that stores transient info*)
	END_VAR
END_FUNCTION

{REDUND_ERROR} FUNCTION vfAddNonEscalatedReactionByName : BOOL (* *) (*$GROUP=User,$CAT=User,$GROUPICON=User.png,$CATICON=User.png*)
	VAR_INPUT
		name : STRING[vfALARMS_MAX_NAME_LEN]; (*The alarm name that triggers these reactions*)
		reactionName1 : STRING[vfALARMS_MAX_REACTION_LEN]; (*A reaction that gets triggered by the associated alarm name*)
		reactionName2 : STRING[vfALARMS_MAX_REACTION_LEN]; (*A reaction that gets triggered by the associated alarm name*)
		reactionName3 : STRING[vfALARMS_MAX_REACTION_LEN]; (*A reaction that gets triggered by the associated alarm name*)
		reactionName4 : STRING[vfALARMS_MAX_REACTION_LEN]; (*A reaction that gets triggered by the associated alarm name*)
		reactionName5 : STRING[vfALARMS_MAX_REACTION_LEN]; (*A reaction that gets triggered by the associated alarm name*)
		reactionName6 : STRING[vfALARMS_MAX_REACTION_LEN]; (*A reaction that gets triggered by the associated alarm name*)
	END_VAR
	VAR_IN_OUT
		data : vfAlarms_Data_typ; (*The VfAlarms data structure that stores transient info*)
	END_VAR
END_FUNCTION

{REDUND_ERROR} FUNCTION vfSetDefaultMapping : BOOL (* *) (*$GROUP=User,$CAT=User,$GROUPICON=User.png,$CATICON=User.png*)
	VAR_INPUT
		type : vfALARMS_MAPPING_enum; (*The default type of mapping to trigger*)
		alarmName : STRING[vfALARMS_MAX_NAME_LEN]; (*The name of the alarm that gets escalated for aggregation mappings*)
	END_VAR
	VAR_IN_OUT
		data : vfAlarms_Data_typ; (*The VfAlarms data structure that stores transient info*)
	END_VAR
END_FUNCTION

{REDUND_ERROR} FUNCTION vfAddAlarm : BOOL (*Add a new alarm definition to the local alarm system*) (*$GROUP=User,$CAT=User,$GROUPICON=User.png,$CATICON=User.png*)
	VAR_INPUT
		name : STRING[vfALARMS_MAX_NAME_LEN]; (*The name of the alarm being defined (i.e. this is the name referenced later by MpAlarmXSet calls)*)
		scope : STRING[vfALARMS_MAX_NAME_LEN]; (*The "Origin" field that will show up on the HMI*)
		code : UDINT; (*The error code associated with this alarm*)
		severity : vfALARMS_SEVERITY_enum; (*The severity of the alarm*)
		behavior : vfALARMS_BEHAVIOR_enum; (*The behavior of the alarm*)
	END_VAR
	VAR_IN_OUT
		data : vfAlarms_Data_typ; (*The VfAlarms data structure that stores transient info*)
	END_VAR
END_FUNCTION

{REDUND_ERROR} FUNCTION vfAddAlarmTextScope : BOOL (*Add a new alarm definition to the local alarm system*) (*$GROUP=User,$CAT=User,$GROUPICON=User.png,$CATICON=User.png*)
	VAR_INPUT
		name : STRING[vfALARMS_MAX_NAME_LEN]; (*The name of the alarm being defined (i.e. this is the name referenced later by MpAlarmXSet calls)*)
		scope : STRING[vfALARMS_MAX_NAME_LEN]; (*The "Origin" field that will show up on the HMI*)
		textScope : STRING[vfALARMS_MAX_NAME_LEN]; (*The "Origin" field that will show up on the HMI*)
		code : UDINT; (*The error code associated with this alarm*)
		severity : vfALARMS_SEVERITY_enum; (*The severity of the alarm*)
		behavior : vfALARMS_BEHAVIOR_enum; (*The behavior of the alarm*)
	END_VAR
	VAR_IN_OUT
		data : vfAlarms_Data_typ; (*The VfAlarms data structure that stores transient info*)
	END_VAR
END_FUNCTION

{REDUND_ERROR} FUNCTION vfCreateAlarmsFaster : BOOL (* *) (*$GROUP=User,$CAT=User,$GROUPICON=User.png,$CATICON=User.png*)
	VAR_IN_OUT
		data : vfAlarms_Data_typ; (*The VfAlarms data structure that stores transient info*)
	END_VAR
END_FUNCTION

{REDUND_ERROR} FUNCTION vfAddLogOriginMapping : BOOL (* *) (*$GROUP=User,$CAT=User,$GROUPICON=User.png,$CATICON=User.png*)
	VAR_INPUT
		originRaw : STRING[32]; (*The default value B&R uses in the "Entered By" column in the Logger*)
		originFormatted : STRING[32]; (*The desired replacement value for the "Entered By" column*)
	END_VAR
	VAR_IN_OUT
		map : Log_Origin_Mappings_typ; (*The global Log mappings data structure*)
	END_VAR
END_FUNCTION

{REDUND_ERROR} FUNCTION vfLookupOrigin : BOOL (* *) (*$GROUP=User,$CAT=User,$GROUPICON=User.png,$CATICON=User.png*)
	VAR_INPUT
		pOriginRaw : UDINT; (*A pointer to the raw "Entered By" name*)
		pOriginFormatted : UDINT; (*A pointer to the new formatted "Entered By" name*)
	END_VAR
	VAR_IN_OUT
		map : Log_Origin_Mappings_typ; (*The global Log mappings data structure*)
	END_VAR
END_FUNCTION

{REDUND_ERROR} FUNCTION vfSetDefaultMappingApi : BOOL (* *) (*$GROUP=User,$CAT=User,$GROUPICON=User.png,$CATICON=User.png*)
	VAR_INPUT
		type : vfALARMS_MAPPING_enum; (*The default type of mapping to trigger*)
		alarmName : vfAlarms_Instance_type; (*The name of the alarm that gets escalated for aggregation mappings*)
	END_VAR
	VAR_IN_OUT
		data : vfAlarms_Data_typ; (*The VfAlarms data structure that stores transient info*)
	END_VAR
END_FUNCTION

{REDUND_ERROR} FUNCTION vfAddAlarmApi : BOOL (*Add a new alarm definition to the local alarm system*) (*$GROUP=User,$CAT=User,$GROUPICON=User.png,$CATICON=User.png*)
	VAR_INPUT
		name : vfAlarms_Instance_type; (*The name of the alarm being defined (i.e. this is the name referenced later by MpAlarmXSet calls)*)
		scope : STRING[vfALARMS_MAX_NAME_LEN]; (*The "Origin" field that will show up on the HMI*)
		code : UDINT; (*The error code associated with this alarm*)
		severity : vfALARMS_SEVERITY_enum; (*The severity of the alarm*)
		behavior : vfALARMS_BEHAVIOR_enum; (*The behavior of the alarm*)
	END_VAR
	VAR_IN_OUT
		data : vfAlarms_Data_typ; (*The VfAlarms data structure that stores transient info*)
	END_VAR
END_FUNCTION

{REDUND_ERROR} FUNCTION vfAddAlarmTextScopeApi : BOOL (*Add a new alarm definition to the local alarm system*) (*$GROUP=User,$CAT=User,$GROUPICON=User.png,$CATICON=User.png*)
	VAR_INPUT
		name : vfAlarms_Instance_type; (*The name of the alarm being defined (i.e. this is the name referenced later by MpAlarmXSet calls)*)
		scope : STRING[vfALARMS_MAX_NAME_LEN]; (*The "Origin" field that will show up on the HMI*)
		textScope : STRING[vfALARMS_MAX_NAME_LEN]; (*The "Origin" field that will show up on the HMI*)
		code : UDINT; (*The error code associated with this alarm*)
		severity : vfALARMS_SEVERITY_enum; (*The severity of the alarm*)
		behavior : vfALARMS_BEHAVIOR_enum; (*The behavior of the alarm*)
	END_VAR
	VAR_IN_OUT
		data : vfAlarms_Data_typ; (*The VfAlarms data structure that stores transient info*)
	END_VAR
END_FUNCTION

{REDUND_ERROR} FUNCTION vfAddAggregationByNameApi : BOOL (* *) (*$GROUP=User,$CAT=User,$GROUPICON=User.png,$CATICON=User.png*)
	VAR_INPUT
		name : STRING[vfALARMS_MAX_NAME_LEN]; (*The alarm name that triggers the aggregation*)
		aggregationName : vfAlarms_Instance_type; (*The name of the alarm that gets escalated during aggregation*)
	END_VAR
	VAR_IN_OUT
		data : vfAlarms_Data_typ; (*The VfAlarms data structure that stores transient info*)
	END_VAR
END_FUNCTION

FUNCTION vfAlarmPersistent : BOOL (*Sets or resets a named alarm based on CurrentState and InstanceID*)
	VAR_INPUT
		alarmComponent : vfAlarms_Component_typ;
		alarm : vfAlarms_Instance_type;
		AlarmConditionActive : BOOL;
	END_VAR
END_FUNCTION

FUNCTION vfAlarmPersistentId : BOOL (*Sets or resets a named alarm based on CurrentState and InstanceID*)
	VAR_INPUT
		alarmComponent : vfAlarms_Component_typ;
		alarm : vfAlarms_Instance_type;
		AlarmConditionActive : BOOL;
	END_VAR
	VAR_IN_OUT
		id : UDINT;
	END_VAR
END_FUNCTION

FUNCTION vfAlarmPersistentSnippetId : BOOL (*Sets or resets a named alarm based on CurrentState and InstanceID*)
	VAR_INPUT
		alarmComponent : vfAlarms_Component_typ;
		alarm : vfAlarms_Instance_type;
		AlarmConditionActive : BOOL;
		snippet : STRING[80];
	END_VAR
	VAR_IN_OUT
		id : UDINT;
	END_VAR
END_FUNCTION

FUNCTION vfAlarmPersistentSnippet : BOOL (*Sets or resets a named alarm based on CurrentState and InstanceID*)
	VAR_INPUT
		alarmComponent : vfAlarms_Component_typ;
		alarm : vfAlarms_Instance_type;
		AlarmConditionActive : BOOL;
		snippet : STRING[80];
	END_VAR
END_FUNCTION

{REDUND_ERROR} FUNCTION vfAlarmEdge : BOOL (*TODO: Add your comment here*) (*$GROUP=User,$CAT=User,$GROUPICON=User.png,$CATICON=User.png*)
	VAR_INPUT
		alarmComponent : vfAlarms_Component_typ;
		alarm : vfAlarms_Instance_type;
	END_VAR
END_FUNCTION

{REDUND_ERROR} FUNCTION vfAlarmEdgeSnippet : BOOL (*TODO: Add your comment here*) (*$GROUP=User,$CAT=User,$GROUPICON=User.png,$CATICON=User.png*)
	VAR_INPUT
		alarmComponent : vfAlarms_Component_typ;
		alarm : vfAlarms_Instance_type;
		snippet : STRING[80];
	END_VAR
END_FUNCTION
```
